LIN {X 0,Y 486.533,Z 891.187,A -85,B 0,C 180,E1 18755.175,E2 18755.175} C_VEL
LIN {X 0,Y 491.243,Z 865.57,A -85,B 0,C 180,E1 18754.171,E2 18754.171} C_VEL
LIN {X 0,Y 494.664,Z 842.648,A -85,B 0,C 180,E1 18753.45,E2 18753.45} C_VEL
LIN {X 0,Y 500.768,Z 797.276,A -85,B 0,C 180,E1 18752.327,E2 18752.327} C_VEL
LIN {X 0,Y 512.182,Z 708.591,A -85,B 0,C 180,E1 18750.377,E2 18750.377} C_VEL
LIN {X 0,Y 521.477,Z 628.395,A -85,B 0,C 180,E1 18748.797,E2 18748.797} C_VEL
LIN {X 0,Y 528.733,Z 554.168,A -85,B 0,C 180,E1 18747.473,E2 18747.473} C_VEL
LIN {X 0,Y 532.171,Z 510.95,A -85,B 0,C 180,E1 18746.749,E2 18746.749} C_VEL
LIN {X 0,Y 523.435,Z 503.495,A -85,B 0,C 180,E1 18744.489,E2 18744.489} C_VEL
LIN {X 0,Y 515.193,Z 497.011,A -85,B 0,C 180,E1 18742.118,E2 18742.118} C_VEL
LIN {X 0,Y 504.103,Z 489.409,A -85,B 0,C 180,E1 18738.384,E2 18738.384} C_VEL
LIN {X 0,Y 494.862,Z 485.329,A -85,B 0,C 180,E1 18734.51,E2 18734.51} C_VEL
LIN {X 0,Y 495.541,Z 486.097,A -85,B 0,C 180,E1 18730.345,E2 18730.345} C_VEL
LIN {X 0,Y 496.003,Z 486.953,A -85,B 0,C 180,E1 18728.93,E2 18728.93} C_VEL
LIN {X 0,Y 497.795,Z 491.194,A -85,B 0,C 180,E1 18724.955,E2 18724.955} C_VEL
LIN {X 0,Y 499.686,Z 495.798,A -85,B 0,C 180,E1 18722.064,E2 18722.064} C_VEL
LIN {X 0,Y 501.598,Z 500.282,A -85,B 0,C 180,E1 18719.772,E2 18719.772} C_VEL
LIN {X 0,Y 504.317,Z 506.652,A -85,B 0,C 180,E1 18717.045,E2 18717.045} C_VEL
LIN {X 0,Y 507.752,Z 515.364,A -85,B 0,C 180,E1 18714.009,E2 18714.009} C_VEL
LIN {X 0,Y 511.515,Z 525.152,A -85,B 0,C 180,E1 18711.116,E2 18711.116} C_VEL
LIN {X 0,Y 512.739,Z 529.148,A -85,B 0,C 180,E1 18710.119,E2 18710.119} C_VEL
LIN {X 0,Y 503.664,Z 561.52,A -85,B 0,C 180,E1 18707.086,E2 18707.086} C_VEL
LIN {X 0,Y 494.519,Z 596.305,A -85,B 0,C 180,E1 18703.918,E2 18703.918} C_VEL
LIN {X 0,Y 488.152,Z 622.653,A -85,B 0,C 180,E1 18701.597,E2 18701.597} C_VEL
LIN {X 0,Y 489.999,Z 648.401,A -85,B 0,C 180,E1 18699.881,E2 18699.881} C_VEL
LIN {X 0,Y 492.993,Z 672.9,A -85,B 0,C 180,E1 18698.025,E2 18698.025} C_VEL
LIN {X 0,Y 496.365,Z 691.421,A -85,B 0,C 180,E1 18696.441,E2 18696.441} C_VEL
LIN {X 0,Y 499.938,Z 706.73,A -85,B 0,C 180,E1 18695.023,E2 18695.023} C_VEL
LIN {X 0,Y 504.478,Z 722.336,A -85,B 0,C 180,E1 18693.452,E2 18693.452} C_VEL
LIN {X 0,Y 511.291,Z 740.682,A -85,B 0,C 180,E1 18691.419,E2 18691.419} C_VEL
LIN {X 0,Y 518.449,Z 755.933,A -85,B 0,C 180,E1 18689.569,E2 18689.569} C_VEL
LIN {X 0,Y 515.516,Z 776.629,A -85,B 0,C 180,E1 18689.383,E2 18689.383} C_VEL
LIN {X 0,Y 510.953,Z 813.16,A -85,B 0,C 180,E1 18688.666,E2 18688.666} C_VEL
LIN {X 0,Y 504.879,Z 851.472,A -85,B 0,C 180,E1 18687.765,E2 18687.765} C_VEL
LIN {X 0,Y 498.91,Z 884.135,A -85,B 0,C 180,E1 18686.793,E2 18686.793} C_VEL
LIN {X 0,Y 492.573,Z 916.172,A -85,B 0,C 180,E1 18685.602,E2 18685.602} C_VEL
LIN {X 0,Y 486.148,Z 946.544,A -85,B 0,C 180,E1 18684.229,E2 18684.229} C_VEL
LIN {X 0,Y 479.406,Z 976.457,A -85,B 0,C 180,E1 18682.618,E2 18682.618} C_VEL
LIN {X 0,Y 472.644,Z 1004.62,A -85,B 0,C 180,E1 18680.832,E2 18680.832} C_VEL
LIN {X 0,Y 466.937,Z 1026.075,A -85,B 0,C 180,E1 18679.222,E2 18679.222} C_VEL
LIN {X 0,Y 460.713,Z 1047.068,A -85,B 0,C 180,E1 18677.366,E2 18677.366} C_VEL
LIN {X 0,Y 454.254,Z 1066.808,A -85,B 0,C 180,E1 18675.311,E2 18675.311} C_VEL
LIN {X 0,Y 447.823,Z 1085.079,A -85,B 0,C 180,E1 18673.094,E2 18673.094} C_VEL
LIN {X 0,Y 441.211,Z 1102.891,A -85,B 0,C 180,E1 18670.57,E2 18670.57} C_VEL
LIN {X 0,Y 434.893,Z 1119.177,A -85,B 0,C 180,E1 18667.868,E2 18667.868} C_VEL
LIN {X 0,Y 428.995,Z 1134.014,A -85,B 0,C 180,E1 18664.983,E2 18664.983} C_VEL
LIN {X 0,Y 423.455,Z 1147.984,A -85,B 0,C 180,E1 18661.771,E2 18661.771} C_VEL
LIN {X 0,Y 418.686,Z 1160.386,A -85,B 0,C 180,E1 18658.373,E2 18658.373} C_VEL
LIN {X 0,Y 414.669,Z 1171.641,A -85,B 0,C 180,E1 18654.653,E2 18654.653} C_VEL
LIN {X 0,Y 411.75,Z 1180.908,A -85,B 0,C 180,E1 18650.912,E2 18650.912} C_VEL
LIN {X 0,Y 409.733,Z 1188.635,A -85,B 0,C 180,E1 18647.026,E2 18647.026} C_VEL
LIN {X 0,Y 408.63,Z 1194.443,A -85,B 0,C 180,E1 18643.296,E2 18643.296} C_VEL
LIN {X 0,Y 408.102,Z 1198.881,A -85,B 0,C 180,E1 18639.446,E2 18639.446} C_VEL
LIN {X 0,Y 407.951,Z 1201.616,A -85,B 0,C 180,E1 18635.907,E2 18635.907} C_VEL
LIN {X 0,Y 407.93,Z 1203.082,A -85,B 0,C 180,E1 18632.386,E2 18632.386} C_VEL
LIN {X 0,Y 407.934,Z 1203.299,A -85,B 0,C 180,E1 18628.875,E2 18628.875} C_VEL
LIN {X 0,Y 407.933,Z 1202.268,A -85,B 0,C 180,E1 18625.359,E2 18625.359} C_VEL
LIN {X 0,Y 408.025,Z 1199.983,A -85,B 0,C 180,E1 18621.827,E2 18621.827} C_VEL
LIN {X 0,Y 408.369,Z 1196.238,A -85,B 0,C 180,E1 18618.129,E2 18618.129} C_VEL
LIN {X 0,Y 409.239,Z 1191.031,A -85,B 0,C 180,E1 18614.408,E2 18614.408} C_VEL
LIN {X 0,Y 410.895,Z 1183.951,A -85,B 0,C 180,E1 18610.524,E2 18610.524} C_VEL
LIN {X 0,Y 413.414,Z 1175.392,A -85,B 0,C 180,E1 18606.78,E2 18606.78} C_VEL
LIN {X 0,Y 416.887,Z 1165.252,A -85,B 0,C 180,E1 18603.155,E2 18603.155} C_VEL
LIN {X 0,Y 421.135,Z 1153.9,A -85,B 0,C 180,E1 18599.777,E2 18599.777} C_VEL
LIN {X 0,Y 426.483,Z 1140.338,A -85,B 0,C 180,E1 18596.405,E2 18596.405} C_VEL
LIN {X 0,Y 432.262,Z 1125.794,A -85,B 0,C 180,E1 18593.358,E2 18593.358} C_VEL
LIN {X 0,Y 438.608,Z 1109.68,A -85,B 0,C 180,E1 18590.502,E2 18590.502} C_VEL
LIN {X 0,Y 444.992,Z 1092.865,A -85,B 0,C 180,E1 18587.962,E2 18587.962} C_VEL
LIN {X 0,Y 451.682,Z 1074.286,A -85,B 0,C 180,E1 18585.561,E2 18585.561} C_VEL
LIN {X 0,Y 458.264,Z 1054.685,A -85,B 0,C 180,E1 18583.399,E2 18583.399} C_VEL
LIN {X 0,Y 464.518,Z 1034.442,A -85,B 0,C 180,E1 18581.488,E2 18581.488} C_VEL
LIN {X 0,Y 470.519,Z 1012.971,A -85,B 0,C 180,E1 18579.766,E2 18579.766} C_VEL
LIN {X 0,Y 476.328,Z 989.375,A -85,B 0,C 180,E1 18578.173,E2 18578.173} C_VEL
LIN {X 0,Y 482.582,Z 962.508,A -85,B 0,C 180,E1 18576.602,E2 18576.602} C_VEL
LIN {X 0,Y 489.045,Z 932.988,A -85,B 0,C 180,E1 18575.131,E2 18575.131} C_VEL
LIN {X 0,Y 495.498,Z 901.478,A -85,B 0,C 180,E1 18573.824,E2 18573.824} C_VEL
LIN {X 0,Y 501.919,Z 867.701,A -85,B 0,C 180,E1 18572.694,E2 18572.694} C_VEL
LIN {X 0,Y 508.145,Z 831.765,A -85,B 0,C 180,E1 18571.754,E2 18571.754} C_VEL
LIN {X 0,Y 513.646,Z 791.804,A -85,B 0,C 180,E1 18570.894,E2 18570.894} C_VEL
LIN {X 0,Y 517.57,Z 753.556,A -85,B 0,C 180,E1 18570.212,E2 18570.212} C_VEL
LIN {X 0,Y 522.49,Z 683.228,A -85,B 0,C 180,E1 18569.21,E2 18569.21} C_VEL
LIN {X 0,Y 524.513,Z 660.576,A -85,B 0,C 180,E1 18568.918,E2 18568.918} C_VEL
LIN {X 0,Y 529.301,Z 622.998,A -85,B 0,C 180,E1 18568.284,E2 18568.284} C_VEL
LIN {X 0,Y 531.877,Z 604.095,A -85,B 0,C 180,E1 18567.995,E2 18567.995} C_VEL
LIN {X 0,Y 536.492,Z 568.871,A -85,B 0,C 180,E1 18567.424,E2 18567.424} C_VEL
LIN {X 0,Y 539.728,Z 546.528,A -85,B 0,C 180,E1 18567.12,E2 18567.12} C_VEL
LIN {X 0,Y 543.093,Z 519.32,A -85,B 0,C 180,E1 18566.641,E2 18566.641} C_VEL
LIN {X 0,Y 533.557,Z 502.875,A -85,B 0,C 180,E1 18563.966,E2 18563.966} C_VEL
LIN {X 0,Y 527.481,Z 493.209,A -85,B 0,C 180,E1 18562.103,E2 18562.103} C_VEL
LIN {X 0,Y 525.221,Z 498.395,A -85,B 0,C 180,E1 18561.814,E2 18561.814} C_VEL
LIN {X 0,Y 519.364,Z 513.075,A -85,B 0,C 180,E1 18561.101,E2 18561.101} C_VEL
LIN {X 0,Y 515.098,Z 522.888,A -85,B 0,C 180,E1 18560.511,E2 18560.511} C_VEL
LIN {X 0,Y 509.416,Z 537.56,A -85,B 0,C 180,E1 18559.776,E2 18559.776} C_VEL
LIN {X 0,Y 505.389,Z 547.114,A -85,B 0,C 180,E1 18559.181,E2 18559.181} C_VEL
LIN {X 0,Y 499.874,Z 561.958,A -85,B 0,C 180,E1 18558.432,E2 18558.432} C_VEL
LIN {X 0,Y 495.743,Z 572.106,A -85,B 0,C 180,E1 18557.78,E2 18557.78} C_VEL
LIN {X 0,Y 490.352,Z 587.299,A -85,B 0,C 180,E1 18557.011,E2 18557.011} C_VEL
LIN {X 0,Y 485.983,Z 598.469,A -85,B 0,C 180,E1 18556.272,E2 18556.272} C_VEL
LIN {X 0,Y 482.289,Z 610.977,A -85,B 0,C 180,E1 18555.674,E2 18555.674} C_VEL
LIN {X 0,Y 478.187,Z 626.414,A -85,B 0,C 180,E1 18554.749,E2 18554.749} C_VEL
LIN {X 0,Y 476.998,Z 630.964,A -85,B 0,C 180,E1 18554.471,E2 18554.471} C_VEL
LIN {X 0,Y 472.235,Z 652.376,A -85,B 0,C 180,E1 18553.476,E2 18553.476} C_VEL
LIN {X 0,Y 468.085,Z 669.271,A -85,B 0,C 180,E1 18552.467,E2 18552.467} C_VEL
LIN {X 0,Y 466.576,Z 674.939,A -85,B 0,C 180,E1 18552.1,E2 18552.1} C_VEL
LIN {X 0,Y 461.683,Z 695.246,A -85,B 0,C 180,E1 18551.113,E2 18551.113} C_VEL
LIN {X 0,Y 457.616,Z 709.605,A -85,B 0,C 180,E1 18550.178,E2 18550.178} C_VEL
LIN {X 0,Y 456.259,Z 714.146,A -85,B 0,C 180,E1 18549.858,E2 18549.858} C_VEL
LIN {X 0,Y 451.518,Z 731.526,A -85,B 0,C 180,E1 18548.959,E2 18548.959} C_VEL
LIN {X 0,Y 447.932,Z 743.114,A -85,B 0,C 180,E1 18548.133,E2 18548.133} C_VEL
LIN {X 0,Y 446.662,Z 747.062,A -85,B 0,C 180,E1 18547.824,E2 18547.824} C_VEL
LIN {X 0,Y 441.934,Z 763.035,A -85,B 0,C 180,E1 18546.936,E2 18546.936} C_VEL
LIN {X 0,Y 438.611,Z 773.144,A -85,B 0,C 180,E1 18546.133,E2 18546.133} C_VEL
LIN {X 0,Y 437.676,Z 775.933,A -85,B 0,C 180,E1 18545.909,E2 18545.909} C_VEL
LIN {X 0,Y 433.17,Z 790.556,A -85,B 0,C 180,E1 18545.049,E2 18545.049} C_VEL
LIN {X 0,Y 430.208,Z 799.346,A -85,B 0,C 180,E1 18544.295,E2 18544.295} C_VEL
LIN {X 0,Y 429.367,Z 801.766,A -85,B 0,C 180,E1 18544.076,E2 18544.076} C_VEL
LIN {X 0,Y 425.227,Z 814.86,A -85,B 0,C 180,E1 18543.286,E2 18543.286} C_VEL
LIN {X 0,Y 422.513,Z 823.016,A -85,B 0,C 180,E1 18542.56,E2 18542.56} C_VEL
LIN {X 0,Y 421.861,Z 825.173,A -85,B 0,C 180,E1 18542.309,E2 18542.309} C_VEL
LIN {X 0,Y 420.52,Z 859.932,A -85,B 0,C 180,E1 18540.647,E2 18540.647} C_VEL
LIN {X 0,Y 418.335,Z 883.831,A -85,B 0,C 180,E1 18539.619,E2 18539.619} C_VEL
LIN {X 0,Y 416.068,Z 978.523,A -85,B 0,C 180,E1 18537.607,E2 18537.607} C_VEL
LIN {X 0,Y 416.149,Z 999.978,A -85,B 0,C 180,E1 18537.078,E2 18537.078} C_VEL
LIN {X 0,Y 416.065,Z 1014.863,A -85,B 0,C 180,E1 18536.487,E2 18536.487} C_VEL
LIN {X 0,Y 415.715,Z 1027.895,A -85,B 0,C 180,E1 18535.724,E2 18535.724} C_VEL
LIN {X 0,Y 415.303,Z 1039.006,A -85,B 0,C 180,E1 18534.889,E2 18534.889} C_VEL
LIN {X 0,Y 414.72,Z 1050.801,A -85,B 0,C 180,E1 18533.771,E2 18533.771} C_VEL
LIN {X 0,Y 413.977,Z 1061.496,A -85,B 0,C 180,E1 18532.446,E2 18532.446} C_VEL
LIN {X 0,Y 413.353,Z 1069.351,A -85,B 0,C 180,E1 18531.234,E2 18531.234} C_VEL
LIN {X 0,Y 412.756,Z 1076.09,A -85,B 0,C 180,E1 18529.955,E2 18529.955} C_VEL
LIN {X 0,Y 412.168,Z 1082.093,A -85,B 0,C 180,E1 18528.526,E2 18528.526} C_VEL
LIN {X 0,Y 411.599,Z 1087.594,A -85,B 0,C 180,E1 18526.8,E2 18526.8} C_VEL
LIN {X 0,Y 411.113,Z 1091.473,A -85,B 0,C 180,E1 18524.916,E2 18524.916} C_VEL
LIN {X 0,Y 410.832,Z 1093.388,A -85,B 0,C 180,E1 18523.31,E2 18523.31} C_VEL
LIN {X 0,Y 410.662,Z 1094.056,A -85,B 0,C 180,E1 18521.694,E2 18521.694} C_VEL
LIN {X 0,Y 410.596,Z 1093.471,A -85,B 0,C 180,E1 18520.053,E2 18520.053} C_VEL
LIN {X 0,Y 410.66,Z 1091.119,A -85,B 0,C 180,E1 18518.077,E2 18518.077} C_VEL
LIN {X 0,Y 410.869,Z 1086.998,A -85,B 0,C 180,E1 18516.212,E2 18516.212} C_VEL
LIN {X 0,Y 411.162,Z 1082.209,A -85,B 0,C 180,E1 18514.659,E2 18514.659} C_VEL
LIN {X 0,Y 411.625,Z 1075.463,A -85,B 0,C 180,E1 18512.983,E2 18512.983} C_VEL
LIN {X 0,Y 412.258,Z 1066.079,A -85,B 0,C 180,E1 18511.219,E2 18511.219} C_VEL
LIN {X 0,Y 412.825,Z 1057.298,A -85,B 0,C 180,E1 18509.909,E2 18509.909} C_VEL
LIN {X 0,Y 413.474,Z 1046.64,A -85,B 0,C 180,E1 18508.613,E2 18508.613} C_VEL
LIN {X 0,Y 414.125,Z 1033.201,A -85,B 0,C 180,E1 18507.341,E2 18507.341} C_VEL
LIN {X 0,Y 414.589,Z 1021.462,A -85,B 0,C 180,E1 18506.475,E2 18506.475} C_VEL
LIN {X 0,Y 414.947,Z 1008.747,A -85,B 0,C 180,E1 18505.745,E2 18505.745} C_VEL
LIN {X 0,Y 415.145,Z 998.499,A -85,B 0,C 180,E1 18505.276,E2 18505.276} C_VEL
LIN {X 0,Y 416.23,Z 998.976,A -85,B 0,C 180,E1 18504.96,E2 18504.96} C_VEL
LIN {X 0,Y 418.224,Z 998.373,A -85,B 0,C 180,E1 18504.649,E2 18504.649} C_VEL
LIN {X 0,Y 421.758,Z 996.071,A -85,B 0,C 180,E1 18504.323,E2 18504.323} C_VEL
LIN {X 0,Y 425.485,Z 994.503,A -85,B 0,C 180,E1 18503.853,E2 18503.853} C_VEL
LIN {X 0,Y 429.216,Z 991.915,A -85,B 0,C 180,E1 18503.555,E2 18503.555} C_VEL
LIN {X 0,Y 433.245,Z 989.836,A -85,B 0,C 180,E1 18503.126,E2 18503.126} C_VEL
LIN {X 0,Y 437.995,Z 986.45,A -85,B 0,C 180,E1 18502.774,E2 18502.774} C_VEL
LIN {X 0,Y 443.74,Z 982.814,A -85,B 0,C 180,E1 18502.273,E2 18502.273} C_VEL
LIN {X 0,Y 448.015,Z 979.633,A -85,B 0,C 180,E1 18501.976,E2 18501.976} C_VEL
LIN {X 0,Y 453.582,Z 975.703,A -85,B 0,C 180,E1 18501.563,E2 18501.563} C_VEL
LIN {X 0,Y 457.655,Z 972.4,A -85,B 0,C 180,E1 18501.328,E2 18501.328} C_VEL
LIN {X 0,Y 464.355,Z 967.489,A -85,B 0,C 180,E1 18500.882,E2 18500.882} C_VEL
LIN {X 0,Y 469.177,Z 963.473,A -85,B 0,C 180,E1 18500.613,E2 18500.613} C_VEL
LIN {X 0,Y 462.39,Z 987.036,A -85,B 0,C 180,E1 18498.735,E2 18498.735} C_VEL
LIN {X 0,Y 455.753,Z 1008.668,A -85,B 0,C 180,E1 18496.752,E2 18496.752} C_VEL
LIN {X 0,Y 448.811,Z 1029.862,A -85,B 0,C 180,E1 18494.481,E2 18494.481} C_VEL
LIN {X 0,Y 442.19,Z 1049.901,A -85,B 0,C 180,E1 18492.016,E2 18492.016} C_VEL
LIN {X 0,Y 435.89,Z 1068.357,A -85,B 0,C 180,E1 18489.371,E2 18489.371} C_VEL
LIN {X 0,Y 430.062,Z 1085.804,A -85,B 0,C 180,E1 18486.528,E2 18486.528} C_VEL
LIN {X 0,Y 424.875,Z 1101.35,A -85,B 0,C 180,E1 18483.577,E2 18483.577} C_VEL
LIN {X 0,Y 420.599,Z 1115.061,A -85,B 0,C 180,E1 18480.617,E2 18480.617} C_VEL
LIN {X 0,Y 416.519,Z 1128.903,A -85,B 0,C 180,E1 18477.138,E2 18477.138} C_VEL
LIN {X 0,Y 413.879,Z 1138.826,A -85,B 0,C 180,E1 18474.25,E2 18474.25} C_VEL
LIN {X 0,Y 411.493,Z 1149.153,A -85,B 0,C 180,E1 18470.781,E2 18470.781} C_VEL
LIN {X 0,Y 409.837,Z 1157.541,A -85,B 0,C 180,E1 18467.318,E2 18467.318} C_VEL
LIN {X 0,Y 408.929,Z 1163.444,A -85,B 0,C 180,E1 18464.387,E2 18464.387} C_VEL
LIN {X 0,Y 407.715,Z 1165.443,A -85,B 0,C 180,E1 18463.346,E2 18463.346} C_VEL
LIN {X 0,Y 400.802,Z 1170.209,A -85,B 0,C 180,E1 18460.402,E2 18460.402} C_VEL
LIN {X 0,Y 400.183,Z 1171.12,A -85,B 0,C 180,E1 18459.621,E2 18459.621} C_VEL
LIN {X 0,Y 400.01,Z 1173.979,A -85,B 0,C 180,E1 18456.749,E2 18456.749} C_VEL
LIN {X 0,Y 399.949,Z 1175.778,A -85,B 0,C 180,E1 18454.016,E2 18454.016} C_VEL
LIN {X 0,Y 399.937,Z 1176.672,A -85,B 0,C 180,E1 18451.291,E2 18451.291} C_VEL
LIN {X 0,Y 399.936,Z 1176.664,A -85,B 0,C 180,E1 18448.569,E2 18448.569} C_VEL
LIN {X 0,Y 399.951,Z 1175.753,A -85,B 0,C 180,E1 18445.844,E2 18445.844} C_VEL
LIN {X 0,Y 400.011,Z 1173.938,A -85,B 0,C 180,E1 18443.111,E2 18443.111} C_VEL
LIN {X 0,Y 400.189,Z 1171.042,A -85,B 0,C 180,E1 18440.22,E2 18440.22} C_VEL
LIN {X 0,Y 400.686,Z 1166.243,A -85,B 0,C 180,E1 18436.713,E2 18436.713} C_VEL
LIN {X 0,Y 401.628,Z 1159.776,A -85,B 0,C 180,E1 18433.216,E2 18433.216} C_VEL
LIN {X 0,Y 402.974,Z 1152.797,A -85,B 0,C 180,E1 18430.12,E2 18430.12} C_VEL
LIN {X 0,Y 404.869,Z 1144.61,A -85,B 0,C 180,E1 18427.035,E2 18427.035} C_VEL
LIN {X 0,Y 408.119,Z 1132.508,A -85,B 0,C 180,E1 18423.207,E2 18423.207} C_VEL
LIN {X 0,Y 411.478,Z 1121.236,A -85,B 0,C 180,E1 18420.171,E2 18420.171} C_VEL
LIN {X 0,Y 416.221,Z 1106.792,A -85,B 0,C 180,E1 18416.792,E2 18416.792} C_VEL
LIN {X 0,Y 421.223,Z 1091.936,A -85,B 0,C 180,E1 18413.812,E2 18413.812} C_VEL
LIN {X 0,Y 426.979,Z 1075.735,A -85,B 0,C 180,E1 18410.957,E2 18410.957} C_VEL
LIN {X 0,Y 433.411,Z 1057.452,A -85,B 0,C 180,E1 18408.188,E2 18408.188} C_VEL
LIN {X 0,Y 439.516,Z 1040.153,A -85,B 0,C 180,E1 18405.885,E2 18405.885} C_VEL
LIN {X 0,Y 446.769,Z 1018.866,A -85,B 0,C 180,E1 18403.431,E2 18403.431} C_VEL
LIN {X 0,Y 453.158,Z 999.494,A -85,B 0,C 180,E1 18401.49,E2 18401.49} C_VEL
LIN {X 0,Y 460.44,Z 976.023,A -85,B 0,C 180,E1 18399.47,E2 18399.47} C_VEL
LIN {X 0,Y 466.465,Z 955.22,A -85,B 0,C 180,E1 18397.928,E2 18397.928} C_VEL
LIN {X 0,Y 473.017,Z 930.366,A -85,B 0,C 180,E1 18396.357,E2 18396.357} C_VEL
LIN {X 0,Y 477.985,Z 909.341,A -85,B 0,C 180,E1 18395.23,E2 18395.23} C_VEL
LIN {X 0,Y 483.181,Z 884.732,A -85,B 0,C 180,E1 18394.112,E2 18394.112} C_VEL
LIN {X 0,Y 487.366,Z 861.137,A -85,B 0,C 180,E1 18393.24,E2 18393.24} C_VEL
LIN {X 0,Y 491.222,Z 835.424,A -85,B 0,C 180,E1 18392.469,E2 18392.469} C_VEL
LIN {X 0,Y 503.581,Z 744.719,A -85,B 0,C 180,E1 18390.359,E2 18390.359} C_VEL
LIN {X 0,Y 513.783,Z 663.571,A -85,B 0,C 180,E1 18388.681,E2 18388.681} C_VEL
LIN {X 0,Y 522.016,Z 587.861,A -85,B 0,C 180,E1 18387.273,E2 18387.273} C_VEL
LIN {X 0,Y 528.229,Z 517.228,A -85,B 0,C 180,E1 18386.077,E2 18386.077} C_VEL
LIN {X 0,Y 528.189,Z 516.76,A -85,B 0,C 180,E1 18386.052,E2 18386.052} C_VEL
LIN {X 0,Y 521.537,Z 511.047,A -85,B 0,C 180,E1 18384.283,E2 18384.283} C_VEL
LIN {X 0,Y 513.386,Z 504.608,A -85,B 0,C 180,E1 18381.899,E2 18381.899} C_VEL
LIN {X 0,Y 502.868,Z 497.289,A -85,B 0,C 180,E1 18378.31,E2 18378.31} C_VEL
LIN {X 0,Y 493.62,Z 493.235,A -85,B 0,C 180,E1 18374.427,E2 18374.427} C_VEL
LIN {X 0,Y 490.745,Z 492.243,A -85,B 0,C 180,E1 18372.951,E2 18372.951} C_VEL
LIN {X 0,Y 491.759,Z 493.451,A -85,B 0,C 180,E1 18369.244,E2 18369.244} C_VEL
LIN {X 0,Y 493.518,Z 497.984,A -85,B 0,C 180,E1 18364.998,E2 18364.998} C_VEL
LIN {X 0,Y 495.306,Z 502.39,A -85,B 0,C 180,E1 18362.198,E2 18362.198} C_VEL
LIN {X 0,Y 497.174,Z 506.879,A -85,B 0,C 180,E1 18359.885,E2 18359.885} C_VEL
LIN {X 0,Y 499.729,Z 512.968,A -85,B 0,C 180,E1 18357.248,E2 18357.248} C_VEL
LIN {X 0,Y 503.08,Z 521.676,A -85,B 0,C 180,E1 18354.182,E2 18354.182} C_VEL
LIN {X 0,Y 506.762,Z 531.481,A -85,B 0,C 180,E1 18351.261,E2 18351.261} C_VEL
LIN {X 0,Y 507.584,Z 534.086,A -85,B 0,C 180,E1 18350.59,E2 18350.59} C_VEL
LIN {X 0,Y 498.418,Z 565.826,A -85,B 0,C 180,E1 18347.605,E2 18347.605} C_VEL
LIN {X 0,Y 488.94,Z 600.817,A -85,B 0,C 180,E1 18344.4,E2 18344.4} C_VEL
LIN {X 0,Y 485.065,Z 616.581,A -85,B 0,C 180,E1 18343.007,E2 18343.007} C_VEL
LIN {X 0,Y 486.674,Z 645.609,A -85,B 0,C 180,E1 18341.089,E2 18341.089} C_VEL
LIN {X 0,Y 488.765,Z 667.497,A -85,B 0,C 180,E1 18339.492,E2 18339.492} C_VEL
LIN {X 0,Y 492.052,Z 689.916,A -85,B 0,C 180,E1 18337.666,E2 18337.666} C_VEL
LIN {X 0,Y 496.427,Z 710.604,A -85,B 0,C 180,E1 18335.755,E2 18335.755} C_VEL
LIN {X 0,Y 501.181,Z 727.72,A -85,B 0,C 180,E1 18334.013,E2 18334.013} C_VEL
LIN {X 0,Y 507.875,Z 746.427,A -85,B 0,C 180,E1 18331.915,E2 18331.915} C_VEL
LIN {X 0,Y 513.758,Z 759.555,A -85,B 0,C 180,E1 18330.311,E2 18330.311} C_VEL
LIN {X 0,Y 510.892,Z 779.529,A -85,B 0,C 180,E1 18330.097,E2 18330.097} C_VEL
LIN {X 0,Y 505.749,Z 818.706,A -85,B 0,C 180,E1 18329.3,E2 18329.3} C_VEL
LIN {X 0,Y 499.219,Z 857.054,A -85,B 0,C 180,E1 18328.363,E2 18328.363} C_VEL
LIN {X 0,Y 492.909,Z 890.183,A -85,B 0,C 180,E1 18327.332,E2 18327.332} C_VEL
LIN {X 0,Y 486.371,Z 922.041,A -85,B 0,C 180,E1 18326.099,E2 18326.099} C_VEL
LIN {X 0,Y 479.461,Z 953.461,A -85,B 0,C 180,E1 18324.624,E2 18324.624} C_VEL
LIN {X 0,Y 472.37,Z 983.55,A -85,B 0,C 180,E1 18322.937,E2 18322.937} C_VEL
LIN {X 0,Y 465.742,Z 1009.903,A -85,B 0,C 180,E1 18321.194,E2 18321.194} C_VEL
LIN {X 0,Y 459.37,Z 1032.171,A -85,B 0,C 180,E1 18319.43,E2 18319.43} C_VEL
LIN {X 0,Y 452.871,Z 1052.669,A -85,B 0,C 180,E1 18317.51,E2 18317.51} C_VEL
LIN {X 0,Y 446.067,Z 1072.391,A -85,B 0,C 180,E1 18315.346,E2 18315.346} C_VEL
LIN {X 0,Y 439.188,Z 1090.996,A -85,B 0,C 180,E1 18312.953,E2 18312.953} C_VEL
LIN {X 0,Y 432.761,Z 1107.475,A -85,B 0,C 180,E1 18310.482,E2 18310.482} C_VEL
LIN {X 0,Y 426.092,Z 1123.874,A -85,B 0,C 180,E1 18307.596,E2 18307.596} C_VEL
LIN {X 0,Y 419.948,Z 1138.652,A -85,B 0,C 180,E1 18304.516,E2 18304.516} C_VEL
LIN {X 0,Y 414.52,Z 1151.912,A -85,B 0,C 180,E1 18301.237,E2 18301.237} C_VEL
LIN {X 0,Y 409.881,Z 1163.689,A -85,B 0,C 180,E1 18297.769,E2 18297.769} C_VEL
LIN {X 0,Y 406.15,Z 1173.986,A -85,B 0,C 180,E1 18294.119,E2 18294.119} C_VEL
LIN {X 0,Y 403.355,Z 1182.79,A -85,B 0,C 180,E1 18290.305,E2 18290.305} C_VEL
LIN {X 0,Y 401.53,Z 1189.848,A -85,B 0,C 180,E1 18286.49,E2 18286.49} C_VEL
LIN {X 0,Y 400.504,Z 1195.302,A -85,B 0,C 180,E1 18282.689,E2 18282.689} C_VEL
LIN {X 0,Y 400.067,Z 1199.269,A -85,B 0,C 180,E1 18278.912,E2 18278.912} C_VEL
LIN {X 0,Y 399.944,Z 1201.754,A -85,B 0,C 180,E1 18275.306,E2 18275.306} C_VEL
LIN {X 0,Y 399.934,Z 1202.969,A -85,B 0,C 180,E1 18271.861,E2 18271.861} C_VEL
LIN {X 0,Y 399.936,Z 1202.996,A -85,B 0,C 180,E1 18268.422,E2 18268.422} C_VEL
LIN {X 0,Y 399.942,Z 1201.821,A -85,B 0,C 180,E1 18264.835,E2 18264.835} C_VEL
LIN {X 0,Y 400.057,Z 1199.39,A -85,B 0,C 180,E1 18261.229,E2 18261.229} C_VEL
LIN {X 0,Y 400.48,Z 1195.481,A -85,B 0,C 180,E1 18257.453,E2 18257.453} C_VEL
LIN {X 0,Y 401.483,Z 1190.086,A -85,B 0,C 180,E1 18253.653,E2 18253.653} C_VEL
LIN {X 0,Y 403.357,Z 1182.785,A -85,B 0,C 180,E1 18249.692,E2 18249.692} C_VEL
LIN {X 0,Y 406.155,Z 1173.978,A -85,B 0,C 180,E1 18245.877,E2 18245.877} C_VEL
LIN {X 0,Y 409.884,Z 1163.678,A -85,B 0,C 180,E1 18242.228,E2 18242.228} C_VEL
LIN {X 0,Y 414.525,Z 1151.898,A -85,B 0,C 180,E1 18238.76,E2 18238.76} C_VEL
LIN {X 0,Y 419.983,Z 1138.549,A -85,B 0,C 180,E1 18235.463,E2 18235.463} C_VEL
LIN {X 0,Y 426.095,Z 1123.839,A -85,B 0,C 180,E1 18232.4,E2 18232.4} C_VEL
LIN {X 0,Y 432.919,Z 1107.068,A -85,B 0,C 180,E1 18229.453,E2 18229.453} C_VEL
LIN {X 0,Y 439.809,Z 1089.346,A -85,B 0,C 180,E1 18226.817,E2 18226.817} C_VEL
LIN {X 0,Y 446.713,Z 1070.541,A -85,B 0,C 180,E1 18224.435,E2 18224.435} C_VEL
LIN {X 0,Y 453.503,Z 1050.665,A -85,B 0,C 180,E1 18222.291,E2 18222.291} C_VEL
LIN {X 0,Y 460.049,Z 1029.72,A -85,B 0,C 180,E1 18220.368,E2 18220.368} C_VEL
LIN {X 0,Y 466.198,Z 1007.987,A -85,B 0,C 180,E1 18218.674,E2 18218.674} C_VEL
LIN {X 0,Y 472.604,Z 982.271,A -85,B 0,C 180,E1 18216.995,E2 18216.995} C_VEL
LIN {X 0,Y 480.508,Z 948.58,A -85,B 0,C 180,E1 18215.134,E2 18215.134} C_VEL
LIN {X 0,Y 487.354,Z 917.154,A -85,B 0,C 180,E1 18213.699,E2 18213.699} C_VEL
LIN {X 0,Y 493.983,Z 884.599,A -85,B 0,C 180,E1 18212.481,E2 18212.481} C_VEL
LIN {X 0,Y 500.295,Z 850.881,A -85,B 0,C 180,E1 18211.477,E2 18211.477} C_VEL
LIN {X 0,Y 506.6,Z 812.409,A -85,B 0,C 180,E1 18210.565,E2 18210.565} C_VEL
LIN {X 0,Y 511.799,Z 770.225,A -85,B 0,C 180,E1 18209.724,E2 18209.724} C_VEL
LIN {X 0,Y 515.455,Z 728.545,A -85,B 0,C 180,E1 18209.06,E2 18209.06} C_VEL
LIN {X 0,Y 519.991,Z 665.837,A -85,B 0,C 180,E1 18208.233,E2 18208.233} C_VEL
LIN {X 0,Y 523.25,Z 637.808,A -85,B 0,C 180,E1 18207.755,E2 18207.755} C_VEL
LIN {X 0,Y 527.822,Z 604.692,A -85,B 0,C 180,E1 18207.252,E2 18207.252} C_VEL
LIN {X 0,Y 532.553,Z 569.137,A -85,B 0,C 180,E1 18206.678,E2 18206.678} C_VEL
LIN {X 0,Y 535.805,Z 546.906,A -85,B 0,C 180,E1 18206.377,E2 18206.377} C_VEL
LIN {X 0,Y 538.738,Z 523.81,A -85,B 0,C 180,E1 18205.977,E2 18205.977} C_VEL
LIN {X 0,Y 529.802,Z 508.232,A -85,B 0,C 180,E1 18203.379,E2 18203.379} C_VEL
LIN {X 0,Y 526.894,Z 503.656,A -85,B 0,C 180,E1 18202.482,E2 18202.482} C_VEL
LIN {X 0,Y 520.808,Z 518.492,A -85,B 0,C 180,E1 18201.749,E2 18201.749} C_VEL
LIN {X 0,Y 517.074,Z 526.968,A -85,B 0,C 180,E1 18201.247,E2 18201.247} C_VEL
LIN {X 0,Y 511.134,Z 542.014,A -85,B 0,C 180,E1 18200.497,E2 18200.497} C_VEL
LIN {X 0,Y 507.188,Z 551.271,A -85,B 0,C 180,E1 18199.934,E2 18199.934} C_VEL
LIN {X 0,Y 501.482,Z 566.318,A -85,B 0,C 180,E1 18199.177,E2 18199.177} C_VEL
LIN {X 0,Y 497.408,Z 576.197,A -85,B 0,C 180,E1 18198.557,E2 18198.557} C_VEL
LIN {X 0,Y 491.817,Z 591.617,A -85,B 0,C 180,E1 18197.779,E2 18197.779} C_VEL
LIN {X 0,Y 487.471,Z 602.573,A -85,B 0,C 180,E1 18197.071,E2 18197.071} C_VEL
LIN {X 0,Y 483.811,Z 614.811,A -85,B 0,C 180,E1 18196.489,E2 18196.489} C_VEL
LIN {X 0,Y 479.476,Z 630.68,A -85,B 0,C 180,E1 18195.544,E2 18195.544} C_VEL
LIN {X 0,Y 478.37,Z 634.918,A -85,B 0,C 180,E1 18195.301,E2 18195.301} C_VEL
LIN {X 0,Y 473.456,Z 656.393,A -85,B 0,C 180,E1 18194.306,E2 18194.306} C_VEL
LIN {X 0,Y 469.127,Z 673.437,A -85,B 0,C 180,E1 18193.293,E2 18193.293} C_VEL
LIN {X 0,Y 467.664,Z 678.834,A -85,B 0,C 180,E1 18192.958,E2 18192.958} C_VEL
LIN {X 0,Y 462.588,Z 699.243,A -85,B 0,C 180,E1 18191.968,E2 18191.968} C_VEL
LIN {X 0,Y 458.259,Z 713.975,A -85,B 0,C 180,E1 18191.013,E2 18191.013} C_VEL
LIN {X 0,Y 456.968,Z 718.237,A -85,B 0,C 180,E1 18190.732,E2 18190.732} C_VEL
LIN {X 0,Y 451.998,Z 735.866,A -85,B 0,C 180,E1 18189.815,E2 18189.815} C_VEL
LIN {X 0,Y 448.177,Z 747.722,A -85,B 0,C 180,E1 18188.969,E2 18188.969} C_VEL
LIN {X 0,Y 447.018,Z 751.288,A -85,B 0,C 180,E1 18188.712,E2 18188.712} C_VEL
LIN {X 0,Y 442.098,Z 767.347,A -85,B 0,C 180,E1 18187.814,E2 18187.814} C_VEL
LIN {X 0,Y 438.48,Z 777.882,A -85,B 0,C 180,E1 18186.975,E2 18186.975} C_VEL
LIN {X 0,Y 436.744,Z 783.34,A -85,B 0,C 180,E1 18186.653,E2 18186.653} C_VEL
LIN {X 0,Y 432.228,Z 797.15,A -85,B 0,C 180,E1 18185.775,E2 18185.775} C_VEL
LIN {X 0,Y 429.109,Z 805.975,A -85,B 0,C 180,E1 18185.005,E2 18185.005} C_VEL
LIN {X 0,Y 424.802,Z 819.185,A -85,B 0,C 180,E1 18184.195,E2 18184.195} C_VEL
LIN {X 0,Y 421.775,Z 827.775,A -85,B 0,C 180,E1 18183.428,E2 18183.428} C_VEL
LIN {X 0,Y 420.968,Z 830.07,A -85,B 0,C 180,E1 18183.221,E2 18183.221} C_VEL
LIN {X 0,Y 416.812,Z 842.6,A -85,B 0,C 180,E1 18182.423,E2 18182.423} C_VEL
LIN {X 0,Y 414.266,Z 849.824,A -85,B 0,C 180,E1 18181.729,E2 18181.729} C_VEL
LIN {X 0,Y 413.752,Z 851.556,A -85,B 0,C 180,E1 18181.523,E2 18181.523} C_VEL
LIN {X 0,Y 412.473,Z 868.78,A -85,B 0,C 180,E1 18180.729,E2 18180.729} C_VEL
LIN {X 0,Y 410.937,Z 885.131,A -85,B 0,C 180,E1 18180.027,E2 18180.027} C_VEL
LIN {X 0,Y 408.524,Z 978.565,A -85,B 0,C 180,E1 18177.979,E2 18177.979} C_VEL
LIN {X 0,Y 408.593,Z 1001.02,A -85,B 0,C 180,E1 18177.418,E2 18177.418} C_VEL
LIN {X 0,Y 408.508,Z 1015.45,A -85,B 0,C 180,E1 18176.843,E2 18176.843} C_VEL
LIN {X 0,Y 408.141,Z 1028.655,A -85,B 0,C 180,E1 18176.067,E2 18176.067} C_VEL
LIN {X 0,Y 407.692,Z 1039.793,A -85,B 0,C 180,E1 18175.217,E2 18175.217} C_VEL
LIN {X 0,Y 407.093,Z 1051.067,A -85,B 0,C 180,E1 18174.134,E2 18174.134} C_VEL
LIN {X 0,Y 406.262,Z 1062.664,A -85,B 0,C 180,E1 18172.692,E2 18172.692} C_VEL
LIN {X 0,Y 405.623,Z 1070.328,A -85,B 0,C 180,E1 18171.494,E2 18171.494} C_VEL
LIN {X 0,Y 404.991,Z 1077.115,A -85,B 0,C 180,E1 18170.191,E2 18170.191} C_VEL
LIN {X 0,Y 404.424,Z 1082.607,A -85,B 0,C 180,E1 18168.881,E2 18168.881} C_VEL
LIN {X 0,Y 403.889,Z 1087.41,A -85,B 0,C 180,E1 18167.417,E2 18167.417} C_VEL
LIN {X 0,Y 403.392,Z 1091.629,A -85,B 0,C 180,E1 18165.648,E2 18165.648} C_VEL
LIN {X 0,Y 402.984,Z 1094.295,A -85,B 0,C 180,E1 18163.717,E2 18163.717} C_VEL
LIN {X 0,Y 402.763,Z 1095.173,A -85,B 0,C 180,E1 18161.96,E2 18161.96} C_VEL
LIN {X 0,Y 402.675,Z 1094.8,A -85,B 0,C 180,E1 18160.414,E2 18160.414} C_VEL
LIN {X 0,Y 402.687,Z 1093.171,A -85,B 0,C 180,E1 18158.745,E2 18158.745} C_VEL
LIN {X 0,Y 402.844,Z 1089.936,A -85,B 0,C 180,E1 18156.91,E2 18156.91} C_VEL
LIN {X 0,Y 403.178,Z 1084.382,A -85,B 0,C 180,E1 18154.907,E2 18154.907} C_VEL
LIN {X 0,Y 403.574,Z 1078.544,A -85,B 0,C 180,E1 18153.356,E2 18153.356} C_VEL
LIN {X 0,Y 404.118,Z 1070.853,A -85,B 0,C 180,E1 18151.745,E2 18151.745} C_VEL
LIN {X 0,Y 404.818,Z 1060.604,A -85,B 0,C 180,E1 18150.07,E2 18150.07} C_VEL
LIN {X 0,Y 405.426,Z 1050.847,A -85,B 0,C 180,E1 18148.807,E2 18148.807} C_VEL
LIN {X 0,Y 406.01,Z 1040.351,A -85,B 0,C 180,E1 18147.696,E2 18147.696} C_VEL
LIN {X 0,Y 406.617,Z 1027.109,A -85,B 0,C 180,E1 18146.576,E2 18146.576} C_VEL
LIN {X 0,Y 407.042,Z 1013.702,A -85,B 0,C 180,E1 18145.732,E2 18145.732} C_VEL
LIN {X 0,Y 407.271,Z 1007.28,A -85,B 0,C 180,E1 18145.364,E2 18145.364} C_VEL
LIN {X 0,Y 408.339,Z 1007.772,A -85,B 0,C 180,E1 18145.041,E2 18145.041} C_VEL
LIN {X 0,Y 410.345,Z 1007.216,A -85,B 0,C 180,E1 18144.717,E2 18144.717} C_VEL
LIN {X 0,Y 413.331,Z 1005.406,A -85,B 0,C 180,E1 18144.423,E2 18144.423} C_VEL
LIN {X 0,Y 416.449,Z 1004.386,A -85,B 0,C 180,E1 18143.967,E2 18143.967} C_VEL
LIN {X 0,Y 420.682,Z 1001.951,A -85,B 0,C 180,E1 18143.544,E2 18143.544} C_VEL
LIN {X 0,Y 425.49,Z 999.583,A -85,B 0,C 180,E1 18143.016,E2 18143.016} C_VEL
LIN {X 0,Y 429.111,Z 997.281,A -85,B 0,C 180,E1 18142.711,E2 18142.711} C_VEL
LIN {X 0,Y 434.263,Z 994.325,A -85,B 0,C 180,E1 18142.232,E2 18142.232} C_VEL
LIN {X 0,Y 438.099,Z 991.701,A -85,B 0,C 180,E1 18141.958,E2 18141.958} C_VEL
LIN {X 0,Y 444.493,Z 987.656,A -85,B 0,C 180,E1 18141.456,E2 18141.456} C_VEL
LIN {X 0,Y 448.406,Z 984.882,A -85,B 0,C 180,E1 18141.2,E2 18141.2} C_VEL
LIN {X 0,Y 455.079,Z 980.187,A -85,B 0,C 180,E1 18140.744,E2 18140.744} C_VEL
LIN {X 0,Y 459.085,Z 977.072,A -85,B 0,C 180,E1 18140.507,E2 18140.507} C_VEL
LIN {X 0,Y 460.312,Z 976.325,A -85,B 0,C 180,E1 18140.411,E2 18140.411} C_VEL
LIN {X 0,Y 452.922,Z 1000.104,A -85,B 0,C 180,E1 18138.356,E2 18138.356} C_VEL
LIN {X 0,Y 446.484,Z 1019.668,A -85,B 0,C 180,E1 18136.389,E2 18136.389} C_VEL
LIN {X 0,Y 439.135,Z 1041.133,A -85,B 0,C 180,E1 18133.896,E2 18133.896} C_VEL
LIN {X 0,Y 433.243,Z 1057.866,A -85,B 0,C 180,E1 18131.659,E2 18131.659} C_VEL
LIN {X 0,Y 426.832,Z 1076.074,A -85,B 0,C 180,E1 18128.89,E2 18128.89} C_VEL
LIN {X 0,Y 421.171,Z 1092.055,A -85,B 0,C 180,E1 18126.071,E2 18126.071} C_VEL
LIN {X 0,Y 415.904,Z 1107.757,A -85,B 0,C 180,E1 18122.912,E2 18122.912} C_VEL
LIN {X 0,Y 411.46,Z 1121.294,A -85,B 0,C 180,E1 18119.72,E2 18119.72} C_VEL
LIN {X 0,Y 408.207,Z 1132.183,A -85,B 0,C 180,E1 18116.79,E2 18116.79} C_VEL
LIN {X 0,Y 405.041,Z 1143.941,A -85,B 0,C 180,E1 18113.112,E2 18113.112} C_VEL
LIN {X 0,Y 403.016,Z 1152.595,A -85,B 0,C 180,E1 18109.872,E2 18109.872} C_VEL
LIN {X 0,Y 401.662,Z 1159.579,A -85,B 0,C 180,E1 18106.786,E2 18106.786} C_VEL
LIN {X 0,Y 400.665,Z 1166.342,A -85,B 0,C 180,E1 18103.128,E2 18103.128} C_VEL
LIN {X 0,Y 400.199,Z 1170.936,A -85,B 0,C 180,E1 18099.783,E2 18099.783} C_VEL
LIN {X 0,Y 400.183,Z 1171.12,A -85,B 0,C 180,E1 18099.621,E2 18099.621} C_VEL
LIN {X 0,Y 399.101,Z 1172.419,A -85,B 0,C 180,E1 18098.534,E2 18098.534} C_VEL
LIN {X 0,Y 392.516,Z 1175.34,A -85,B 0,C 180,E1 18095.459,E2 18095.459} C_VEL
LIN {X 0,Y 391.961,Z 1175.77,A -85,B 0,C 180,E1 18094.65,E2 18094.65} C_VEL
LIN {X 0,Y 391.94,Z 1176.887,A -85,B 0,C 180,E1 18091.61,E2 18091.61} C_VEL
LIN {X 0,Y 391.94,Z 1176.973,A -85,B 0,C 180,E1 18088.832,E2 18088.832} C_VEL
LIN {X 0,Y 391.955,Z 1176.149,A -85,B 0,C 180,E1 18086.052,E2 18086.052} C_VEL
LIN {X 0,Y 392.015,Z 1174.416,A -85,B 0,C 180,E1 18083.264,E2 18083.264} C_VEL
LIN {X 0,Y 392.178,Z 1171.766,A -85,B 0,C 180,E1 18080.463,E2 18080.463} C_VEL
LIN {X 0,Y 392.553,Z 1167.971,A -85,B 0,C 180,E1 18077.498,E2 18077.498} C_VEL
LIN {X 0,Y 393.38,Z 1162.34,A -85,B 0,C 180,E1 18074.069,E2 18074.069} C_VEL
LIN {X 0,Y 394.907,Z 1154.448,A -85,B 0,C 180,E1 18070.323,E2 18070.323} C_VEL
LIN {X 0,Y 396.813,Z 1146.443,A -85,B 0,C 180,E1 18067.169,E2 18067.169} C_VEL
LIN {X 0,Y 399.515,Z 1136.681,A -85,B 0,C 180,E1 18063.868,E2 18063.868} C_VEL
LIN {X 0,Y 403.385,Z 1124.122,A -85,B 0,C 180,E1 18060.283,E2 18060.283} C_VEL
LIN {X 0,Y 407.383,Z 1112.126,A -85,B 0,C 180,E1 18057.321,E2 18057.321} C_VEL
LIN {X 0,Y 412.723,Z 1097.218,A -85,B 0,C 180,E1 18054.109,E2 18054.109} C_VEL
LIN {X 0,Y 418.484,Z 1081.289,A -85,B 0,C 180,E1 18051.162,E2 18051.162} C_VEL
LIN {X 0,Y 425.143,Z 1063.453,A -85,B 0,C 180,E1 18048.276,E2 18048.276} C_VEL
LIN {X 0,Y 431.83,Z 1045.088,A -85,B 0,C 180,E1 18045.727,E2 18045.727} C_VEL
LIN {X 0,Y 439.055,Z 1025.214,A -85,B 0,C 180,E1 18043.316,E2 18043.316} C_VEL
LIN {X 0,Y 446.158,Z 1004.37,A -85,B 0,C 180,E1 18041.151,E2 18041.151} C_VEL
LIN {X 0,Y 453.365,Z 982.514,A -85,B 0,C 180,E1 18039.178,E2 18039.178} C_VEL
LIN {X 0,Y 459.974,Z 960.546,A -85,B 0,C 180,E1 18037.493,E2 18037.493} C_VEL
LIN {X 0,Y 465.884,Z 939.59,A -85,B 0,C 180,E1 18036.098,E2 18036.098} C_VEL
LIN {X 0,Y 471.97,Z 915.203,A -85,B 0,C 180,E1 18034.719,E2 18034.719} C_VEL
LIN {X 0,Y 476.936,Z 893.107,A -85,B 0,C 180,E1 18033.668,E2 18033.668} C_VEL
LIN {X 0,Y 482.012,Z 866.564,A -85,B 0,C 180,E1 18032.63,E2 18032.63} C_VEL
LIN {X 0,Y 485.41,Z 845.118,A -85,B 0,C 180,E1 18031.951,E2 18031.951} C_VEL
LIN {X 0,Y 492.444,Z 796.283,A -85,B 0,C 180,E1 18030.727,E2 18030.727} C_VEL
LIN {X 0,Y 504.375,Z 709.08,A -85,B 0,C 180,E1 18028.799,E2 18028.799} C_VEL
LIN {X 0,Y 513.868,Z 631.384,A -85,B 0,C 180,E1 18027.266,E2 18027.266} C_VEL
LIN {X 0,Y 521.367,Z 558.159,A -85,B 0,C 180,E1 18025.962,E2 18025.962} C_VEL
LIN {X 0,Y 524.291,Z 522.66,A -85,B 0,C 180,E1 18025.35,E2 18025.35} C_VEL
LIN {X 0,Y 519.452,Z 518.461,A -85,B 0,C 180,E1 18024.024,E2 18024.024} C_VEL
LIN {X 0,Y 511.758,Z 512.303,A -85,B 0,C 180,E1 18021.731,E2 18021.731} C_VEL
LIN {X 0,Y 501.337,Z 505.068,A -85,B 0,C 180,E1 18018.128,E2 18018.128} C_VEL
LIN {X 0,Y 492.43,Z 501.144,A -85,B 0,C 180,E1 18014.343,E2 18014.343} C_VEL
LIN {X 0,Y 486.882,Z 499.43,A -85,B 0,C 180,E1 18011.251,E2 18011.251} C_VEL
LIN {X 0,Y 487.554,Z 500.477,A -85,B 0,C 180,E1 18009.086,E2 18009.086} C_VEL
LIN {X 0,Y 489.242,Z 504.773,A -85,B 0,C 180,E1 18005.042,E2 18005.042} C_VEL
LIN {X 0,Y 490.929,Z 508.983,A -85,B 0,C 180,E1 18002.335,E2 18002.335} C_VEL
LIN {X 0,Y 492.752,Z 513.476,A -85,B 0,C 180,E1 18000,E2 18000} C_VEL
LIN {X 0,Y 495.247,Z 519.597,A -85,B 0,C 180,E1 17997.338,E2 17997.338} C_VEL
LIN {X 0,Y 498.679,Z 528.684,A -85,B 0,C 180,E1 17994.131,E2 17994.131} C_VEL
LIN {X 0,Y 502.304,Z 538.629,A -85,B 0,C 180,E1 17991.183,E2 17991.183} C_VEL
LIN {X 0,Y 502.447,Z 539.047,A -85,B 0,C 180,E1 17991.07,E2 17991.07} C_VEL
LIN {X 0,Y 493.205,Z 570.161,A -85,B 0,C 180,E1 17988.131,E2 17988.131} C_VEL
LIN {X 0,Y 483.535,Z 604.807,A -85,B 0,C 180,E1 17984.94,E2 17984.94} C_VEL
LIN {X 0,Y 482.24,Z 610.539,A -85,B 0,C 180,E1 17984.447,E2 17984.447} C_VEL
LIN {X 0,Y 484.014,Z 649.87,A -85,B 0,C 180,E1 17981.824,E2 17981.824} C_VEL
LIN {X 0,Y 485.94,Z 671.768,A -85,B 0,C 180,E1 17980.215,E2 17980.215} C_VEL
LIN {X 0,Y 489.058,Z 694.545,A -85,B 0,C 180,E1 17978.344,E2 17978.344} C_VEL
LIN {X 0,Y 493.301,Z 715.728,A -85,B 0,C 180,E1 17976.368,E2 17976.368} C_VEL
LIN {X 0,Y 497.896,Z 733.215,A -85,B 0,C 180,E1 17974.563,E2 17974.563} C_VEL
LIN {X 0,Y 504.414,Z 752.155,A -85,B 0,C 180,E1 17972.412,E2 17972.412} C_VEL
LIN {X 0,Y 509.136,Z 763.083,A -85,B 0,C 180,E1 17971.059,E2 17971.059} C_VEL
LIN {X 0,Y 506.205,Z 783.812,A -85,B 0,C 180,E1 17970.798,E2 17970.798} C_VEL
LIN {X 0,Y 500.513,Z 823.972,A -85,B 0,C 180,E1 17969.945,E2 17969.945} C_VEL
LIN {X 0,Y 493.921,Z 861.128,A -85,B 0,C 180,E1 17969.014,E2 17969.014} C_VEL
LIN {X 0,Y 487.423,Z 893.882,A -85,B 0,C 180,E1 17967.962,E2 17967.962} C_VEL
LIN {X 0,Y 480.764,Z 925.114,A -85,B 0,C 180,E1 17966.724,E2 17966.724} C_VEL
LIN {X 0,Y 473.566,Z 956.555,A -85,B 0,C 180,E1 17965.215,E2 17965.215} C_VEL
LIN {X 0,Y 466.084,Z 987.317,A -85,B 0,C 180,E1 17963.454,E2 17963.454} C_VEL
LIN {X 0,Y 460.004,Z 1010.548,A -85,B 0,C 180,E1 17961.89,E2 17961.89} C_VEL
LIN {X 0,Y 453.676,Z 1032.047,A -85,B 0,C 180,E1 17960.179,E2 17960.179} C_VEL
LIN {X 0,Y 446.744,Z 1053.159,A -85,B 0,C 180,E1 17958.182,E2 17958.182} C_VEL
LIN {X 0,Y 439.972,Z 1072.039,A -85,B 0,C 180,E1 17956.086,E2 17956.086} C_VEL
LIN {X 0,Y 432.871,Z 1090.592,A -85,B 0,C 180,E1 17953.679,E2 17953.679} C_VEL
LIN {X 0,Y 425.978,Z 1107.654,A -85,B 0,C 180,E1 17951.087,E2 17951.087} C_VEL
LIN {X 0,Y 419.405,Z 1123.31,A -85,B 0,C 180,E1 17948.303,E2 17948.303} C_VEL
LIN {X 0,Y 413.001,Z 1138.189,A -85,B 0,C 180,E1 17945.181,E2 17945.181} C_VEL
LIN {X 0,Y 407.115,Z 1152.054,A -85,B 0,C 180,E1 17941.706,E2 17941.706} C_VEL
LIN {X 0,Y 402.287,Z 1163.79,A -85,B 0,C 180,E1 17938.178,E2 17938.178} C_VEL
LIN {X 0,Y 398.408,Z 1174.048,A -85,B 0,C 180,E1 17934.46,E2 17934.46} C_VEL
LIN {X 0,Y 395.494,Z 1182.821,A -85,B 0,C 180,E1 17930.572,E2 17930.572} C_VEL
LIN {X 0,Y 393.587,Z 1189.83,A -85,B 0,C 180,E1 17926.681,E2 17926.681} C_VEL
LIN {X 0,Y 392.522,Z 1195.234,A -85,B 0,C 180,E1 17922.802,E2 17922.802} C_VEL
LIN {X 0,Y 392.069,Z 1199.142,A -85,B 0,C 180,E1 17918.948,E2 17918.948} C_VEL
LIN {X 0,Y 391.946,Z 1201.564,A -85,B 0,C 180,E1 17915.268,E2 17915.268} C_VEL
LIN {X 0,Y 391.938,Z 1202.72,A -85,B 0,C 180,E1 17911.752,E2 17911.752} C_VEL
LIN {X 0,Y 391.939,Z 1202.72,A -85,B 0,C 180,E1 17908.244,E2 17908.244} C_VEL
LIN {X 0,Y 391.946,Z 1201.564,A -85,B 0,C 180,E1 17904.729,E2 17904.729} C_VEL
LIN {X 0,Y 392.068,Z 1199.141,A -85,B 0,C 180,E1 17901.049,E2 17901.049} C_VEL
LIN {X 0,Y 392.522,Z 1195.232,A -85,B 0,C 180,E1 17897.194,E2 17897.194} C_VEL
LIN {X 0,Y 393.601,Z 1189.769,A -85,B 0,C 180,E1 17893.28,E2 17893.28} C_VEL
LIN {X 0,Y 395.496,Z 1182.811,A -85,B 0,C 180,E1 17889.424,E2 17889.424} C_VEL
LIN {X 0,Y 398.412,Z 1174.037,A -85,B 0,C 180,E1 17885.536,E2 17885.536} C_VEL
LIN {X 0,Y 402.289,Z 1163.775,A -85,B 0,C 180,E1 17881.818,E2 17881.818} C_VEL
LIN {X 0,Y 407.118,Z 1152.031,A -85,B 0,C 180,E1 17878.291,E2 17878.291} C_VEL
LIN {X 0,Y 413.004,Z 1138.156,A -85,B 0,C 180,E1 17874.815,E2 17874.815} C_VEL
LIN {X 0,Y 419.53,Z 1123.006,A -85,B 0,C 180,E1 17871.64,E2 17871.64} C_VEL
LIN {X 0,Y 426.333,Z 1106.795,A -85,B 0,C 180,E1 17868.772,E2 17868.772} C_VEL
LIN {X 0,Y 433.385,Z 1089.259,A -85,B 0,C 180,E1 17866.134,E2 17866.134} C_VEL
LIN {X 0,Y 440.55,Z 1070.421,A -85,B 0,C 180,E1 17863.724,E2 17863.724} C_VEL
LIN {X 0,Y 447.612,Z 1050.472,A -85,B 0,C 180,E1 17861.552,E2 17861.552} C_VEL
LIN {X 0,Y 454.359,Z 1029.657,A -85,B 0,C 180,E1 17859.624,E2 17859.624} C_VEL
LIN {X 0,Y 460.757,Z 1007.822,A -85,B 0,C 180,E1 17857.912,E2 17857.912} C_VEL
LIN {X 0,Y 467.085,Z 983.17,A -85,B 0,C 180,E1 17856.294,E2 17856.294} C_VEL
LIN {X 0,Y 474.856,Z 951.069,A -85,B 0,C 180,E1 17854.502,E2 17854.502} C_VEL
LIN {X 0,Y 481.91,Z 919.615,A -85,B 0,C 180,E1 17853.044,E2 17853.044} C_VEL
LIN {X 0,Y 488.815,Z 886.816,A -85,B 0,C 180,E1 17851.796,E2 17851.796} C_VEL
LIN {X 0,Y 495.439,Z 852.746,A -85,B 0,C 180,E1 17850.763,E2 17850.763} C_VEL
LIN {X 0,Y 502.168,Z 812.982,A -85,B 0,C 180,E1 17849.812,E2 17849.812} C_VEL
LIN {X 0,Y 507.269,Z 773.74,A -85,B 0,C 180,E1 17849.015,E2 17849.015} C_VEL
LIN {X 0,Y 511.245,Z 732.69,A -85,B 0,C 180,E1 17848.336,E2 17848.336} C_VEL
LIN {X 0,Y 516.148,Z 666.708,A -85,B 0,C 180,E1 17847.461,E2 17847.461} C_VEL
LIN {X 0,Y 517.624,Z 650.639,A -85,B 0,C 180,E1 17847.205,E2 17847.205} C_VEL
LIN {X 0,Y 523.21,Z 610.685,A -85,B 0,C 180,E1 17846.6,E2 17846.6} C_VEL
LIN {X 0,Y 527.875,Z 575.078,A -85,B 0,C 180,E1 17846,E2 17846} C_VEL
LIN {X 0,Y 531.975,Z 547.261,A -85,B 0,C 180,E1 17845.623,E2 17845.623} C_VEL
LIN {X 0,Y 534.373,Z 528.199,A -85,B 0,C 180,E1 17845.281,E2 17845.281} C_VEL
LIN {X 0,Y 526.486,Z 514.24,A -85,B 0,C 180,E1 17842.904,E2 17842.904} C_VEL
LIN {X 0,Y 520.196,Z 528.47,A -85,B 0,C 180,E1 17842.107,E2 17842.107} C_VEL
LIN {X 0,Y 512.85,Z 546.662,A -85,B 0,C 180,E1 17841.203,E2 17841.203} C_VEL
LIN {X 0,Y 509.123,Z 555.288,A -85,B 0,C 180,E1 17840.687,E2 17840.687} C_VEL
LIN {X 0,Y 503.17,Z 570.688,A -85,B 0,C 180,E1 17839.917,E2 17839.917} C_VEL
LIN {X 0,Y 499.16,Z 580.29,A -85,B 0,C 180,E1 17839.328,E2 17839.328} C_VEL
LIN {X 0,Y 493.351,Z 595.984,A -85,B 0,C 180,E1 17838.539,E2 17838.539} C_VEL
LIN {X 0,Y 489.121,Z 606.47,A -85,B 0,C 180,E1 17837.872,E2 17837.872} C_VEL
LIN {X 0,Y 485.443,Z 618.591,A -85,B 0,C 180,E1 17837.3,E2 17837.3} C_VEL
LIN {X 0,Y 480.914,Z 634.75,A -85,B 0,C 180,E1 17836.348,E2 17836.348} C_VEL
LIN {X 0,Y 479.751,Z 639.271,A -85,B 0,C 180,E1 17836.11,E2 17836.11} C_VEL
LIN {X 0,Y 474.617,Z 661.054,A -85,B 0,C 180,E1 17835.097,E2 17835.097} C_VEL
LIN {X 0,Y 470.085,Z 678.192,A -85,B 0,C 180,E1 17834.074,E2 17834.074} C_VEL
LIN {X 0,Y 468.819,Z 682.878,A -85,B 0,C 180,E1 17833.804,E2 17833.804} C_VEL
LIN {X 0,Y 463.533,Z 703.43,A -85,B 0,C 180,E1 17832.809,E2 17832.809} C_VEL
LIN {X 0,Y 459.002,Z 718.307,A -85,B 0,C 180,E1 17831.848,E2 17831.848} C_VEL
LIN {X 0,Y 457.777,Z 722.35,A -85,B 0,C 180,E1 17831.601,E2 17831.601} C_VEL
LIN {X 0,Y 452.582,Z 740.187,A -85,B 0,C 180,E1 17830.671,E2 17830.671} C_VEL
LIN {X 0,Y 448.5,Z 752.376,A -85,B 0,C 180,E1 17829.799,E2 17829.799} C_VEL
LIN {X 0,Y 447.236,Z 756.325,A -85,B 0,C 180,E1 17829.558,E2 17829.558} C_VEL
LIN {X 0,Y 442.16,Z 772.27,A -85,B 0,C 180,E1 17828.649,E2 17828.649} C_VEL
LIN {X 0,Y 437.986,Z 784.06,A -85,B 0,C 180,E1 17827.741,E2 17827.741} C_VEL
LIN {X 0,Y 432.988,Z 799.08,A -85,B 0,C 180,E1 17826.846,E2 17826.846} C_VEL
LIN {X 0,Y 429.415,Z 808.79,A -85,B 0,C 180,E1 17826.015,E2 17826.015} C_VEL
LIN {X 0,Y 424.524,Z 823.233,A -85,B 0,C 180,E1 17825.127,E2 17825.127} C_VEL
LIN {X 0,Y 421.149,Z 832.461,A -85,B 0,C 180,E1 17824.307,E2 17824.307} C_VEL
LIN {X 0,Y 415.752,Z 848.052,A -85,B 0,C 180,E1 17823.257,E2 17823.257} C_VEL
LIN {X 0,Y 413.019,Z 855.344,A -85,B 0,C 180,E1 17822.515,E2 17822.515} C_VEL
LIN {X 0,Y 407.522,Z 871.306,A -85,B 0,C 180,E1 17821.547,E2 17821.547} C_VEL
LIN {X 0,Y 404.399,Z 880.105,A -85,B 0,C 180,E1 17820.779,E2 17820.779} C_VEL
LIN {X 0,Y 403.987,Z 881.583,A -85,B 0,C 180,E1 17820.641,E2 17820.641} C_VEL
LIN {X 0,Y 403.535,Z 887.725,A -85,B 0,C 180,E1 17820.426,E2 17820.426} C_VEL
LIN {X 0,Y 400.989,Z 981.142,A -85,B 0,C 180,E1 17818.312,E2 17818.312} C_VEL
LIN {X 0,Y 401.05,Z 1002.749,A -85,B 0,C 180,E1 17817.75,E2 17817.75} C_VEL
LIN {X 0,Y 400.936,Z 1017.415,A -85,B 0,C 180,E1 17817.141,E2 17817.141} C_VEL
LIN {X 0,Y 400.538,Z 1030.438,A -85,B 0,C 180,E1 17816.35,E2 17816.35} C_VEL
LIN {X 0,Y 400.067,Z 1041.488,A -85,B 0,C 180,E1 17815.485,E2 17815.485} C_VEL
LIN {X 0,Y 399.405,Z 1053.194,A -85,B 0,C 180,E1 17814.331,E2 17814.331} C_VEL
LIN {X 0,Y 398.565,Z 1063.993,A -85,B 0,C 180,E1 17812.939,E2 17812.939} C_VEL
LIN {X 0,Y 397.91,Z 1071.353,A -85,B 0,C 180,E1 17811.765,E2 17811.765} C_VEL
LIN {X 0,Y 397.234,Z 1078.145,A -85,B 0,C 180,E1 17810.437,E2 17810.437} C_VEL
LIN {X 0,Y 396.572,Z 1084.222,A -85,B 0,C 180,E1 17808.953,E2 17808.953} C_VEL
LIN {X 0,Y 395.925,Z 1089.792,A -85,B 0,C 180,E1 17807.159,E2 17807.159} C_VEL
LIN {X 0,Y 395.369,Z 1093.729,A -85,B 0,C 180,E1 17805.201,E2 17805.201} C_VEL
LIN {X 0,Y 395.039,Z 1095.653,A -85,B 0,C 180,E1 17803.532,E2 17803.532} C_VEL
LIN {X 0,Y 394.849,Z 1096.316,A -85,B 0,C 180,E1 17802.004,E2 17802.004} C_VEL
LIN {X 0,Y 394.749,Z 1095.84,A -85,B 0,C 180,E1 17800.313,E2 17800.313} C_VEL
LIN {X 0,Y 394.767,Z 1094.1,A -85,B 0,C 180,E1 17798.609,E2 17798.609} C_VEL
LIN {X 0,Y 394.963,Z 1090.374,A -85,B 0,C 180,E1 17796.58,E2 17796.58} C_VEL
LIN {X 0,Y 395.29,Z 1084.948,A -85,B 0,C 180,E1 17794.692,E2 17794.692} C_VEL
LIN {X 0,Y 395.713,Z 1078.956,A -85,B 0,C 180,E1 17793.109,E2 17793.109} C_VEL
LIN {X 0,Y 396.339,Z 1070.543,A -85,B 0,C 180,E1 17791.358,E2 17791.358} C_VEL
LIN {X 0,Y 397.025,Z 1060.456,A -85,B 0,C 180,E1 17789.751,E2 17789.751} C_VEL
LIN {X 0,Y 397.666,Z 1050.454,A -85,B 0,C 180,E1 17788.466,E2 17788.466} C_VEL
LIN {X 0,Y 398.374,Z 1037.942,A -85,B 0,C 180,E1 17787.17,E2 17787.17} C_VEL
LIN {X 0,Y 398.926,Z 1024.903,A -85,B 0,C 180,E1 17786.142,E2 17786.142} C_VEL
LIN {X 0,Y 399.25,Z 1015.282,A -85,B 0,C 180,E1 17785.528,E2 17785.528} C_VEL
LIN {X 0,Y 400.546,Z 1015.792,A -85,B 0,C 180,E1 17785.134,E2 17785.134} C_VEL
LIN {X 0,Y 402.558,Z 1015.211,A -85,B 0,C 180,E1 17784.813,E2 17784.813} C_VEL
LIN {X 0,Y 404.938,Z 1014.067,A -85,B 0,C 180,E1 17784.53,E2 17784.53} C_VEL
LIN {X 0,Y 408.335,Z 1013.064,A -85,B 0,C 180,E1 17784.007,E2 17784.007} C_VEL
LIN {X 0,Y 411.646,Z 1011.333,A -85,B 0,C 180,E1 17783.653,E2 17783.653} C_VEL
LIN {X 0,Y 416.222,Z 1009.464,A -85,B 0,C 180,E1 17783.089,E2 17783.089} C_VEL
LIN {X 0,Y 419.658,Z 1007.615,A -85,B 0,C 180,E1 17782.757,E2 17782.757} C_VEL
LIN {X 0,Y 425.542,Z 1004.611,A -85,B 0,C 180,E1 17782.174,E2 17782.174} C_VEL
LIN {X 0,Y 429.15,Z 1002.517,A -85,B 0,C 180,E1 17781.871,E2 17781.871} C_VEL
LIN {X 0,Y 435.442,Z 998.785,A -85,B 0,C 180,E1 17781.348,E2 17781.348} C_VEL
LIN {X 0,Y 439.188,Z 996.386,A -85,B 0,C 180,E1 17781.07,E2 17781.07} C_VEL
LIN {X 0,Y 445.822,Z 992.012,A -85,B 0,C 180,E1 17780.601,E2 17780.601} C_VEL
LIN {X 0,Y 451.387,Z 988.344,A -85,B 0,C 180,E1 17780.226,E2 17780.226} C_VEL
LIN {X 0,Y 444.818,Z 1008.319,A -85,B 0,C 180,E1 17778.368,E2 17778.368} C_VEL
LIN {X 0,Y 437.096,Z 1030.39,A -85,B 0,C 180,E1 17775.99,E2 17775.99} C_VEL
LIN {X 0,Y 430.313,Z 1049.208,A -85,B 0,C 180,E1 17773.641,E2 17773.641} C_VEL
LIN {X 0,Y 423.264,Z 1068.33,A -85,B 0,C 180,E1 17770.873,E2 17770.873} C_VEL
LIN {X 0,Y 417.322,Z 1084.496,A -85,B 0,C 180,E1 17768.183,E2 17768.183} C_VEL
LIN {X 0,Y 411.037,Z 1101.722,A -85,B 0,C 180,E1 17764.868,E2 17764.868} C_VEL
LIN {X 0,Y 406.418,Z 1114.964,A -85,B 0,C 180,E1 17761.92,E2 17761.92} C_VEL
LIN {X 0,Y 401.732,Z 1129.266,A -85,B 0,C 180,E1 17758.224,E2 17758.224} C_VEL
LIN {X 0,Y 398.636,Z 1139.633,A -85,B 0,C 180,E1 17755.083,E2 17755.083} C_VEL
LIN {X 0,Y 396.072,Z 1149.477,A -85,B 0,C 180,E1 17751.63,E2 17751.63} C_VEL
LIN {X 0,Y 394.116,Z 1158.23,A -85,B 0,C 180,E1 17747.879,E2 17747.879} C_VEL
LIN {X 0,Y 393.085,Z 1164.066,A -85,B 0,C 180,E1 17744.848,E2 17744.848} C_VEL
LIN {X 0,Y 392.463,Z 1168.683,A -85,B 0,C 180,E1 17741.911,E2 17741.911} C_VEL
LIN {X 0,Y 392.137,Z 1172.482,A -85,B 0,C 180,E1 17738.802,E2 17738.802} C_VEL
LIN {X 0,Y 391.976,Z 1175.545,A -85,B 0,C 180,E1 17735.124,E2 17735.124} C_VEL
LIN {X 0,Y 391.961,Z 1175.77,A -85,B 0,C 180,E1 17734.65,E2 17734.65} C_VEL
LIN {X 0,Y 390.949,Z 1176.35,A -85,B 0,C 180,E1 17733.527,E2 17733.527} C_VEL
LIN {X 0,Y 386.667,Z 1177.167,A -85,B 0,C 180,E1 17731.564,E2 17731.564} C_VEL
LIN {X 0,Y 384.145,Z 1177.402,A -85,B 0,C 180,E1 17730.025,E2 17730.025} C_VEL
LIN {X 0,Y 383.938,Z 1177.349,A -85,B 0,C 180,E1 17729.525,E2 17729.525} C_VEL
LIN {X 0,Y 383.959,Z 1176.547,A -85,B 0,C 180,E1 17726.269,E2 17726.269} C_VEL
LIN {X 0,Y 384.022,Z 1174.783,A -85,B 0,C 180,E1 17723.273,E2 17723.273} C_VEL
LIN {X 0,Y 384.193,Z 1172.172,A -85,B 0,C 180,E1 17720.414,E2 17720.414} C_VEL
LIN {X 0,Y 384.588,Z 1168.415,A -85,B 0,C 180,E1 17717.388,E2 17717.388} C_VEL
LIN {X 0,Y 385.357,Z 1163.346,A -85,B 0,C 180,E1 17714.192,E2 17714.192} C_VEL
LIN {X 0,Y 387.044,Z 1155.124,A -85,B 0,C 180,E1 17710.113,E2 17710.113} C_VEL
LIN {X 0,Y 389.068,Z 1147.06,A -85,B 0,C 180,E1 17706.848,E2 17706.848} C_VEL
LIN {X 0,Y 391.907,Z 1137.359,A -85,B 0,C 180,E1 17703.484,E2 17703.484} C_VEL
LIN {X 0,Y 395.955,Z 1124.892,A -85,B 0,C 180,E1 17699.835,E2 17699.835} C_VEL
LIN {X 0,Y 400.142,Z 1112.969,A -85,B 0,C 180,E1 17696.824,E2 17696.824} C_VEL
LIN {X 0,Y 405.699,Z 1098.164,A -85,B 0,C 180,E1 17693.564,E2 17693.564} C_VEL
LIN {X 0,Y 411.737,Z 1082.215,A -85,B 0,C 180,E1 17690.557,E2 17690.557} C_VEL
LIN {X 0,Y 418.603,Z 1064.615,A -85,B 0,C 180,E1 17687.658,E2 17687.658} C_VEL
LIN {X 0,Y 425.525,Z 1046.361,A -85,B 0,C 180,E1 17685.084,E2 17685.084} C_VEL
LIN {X 0,Y 432.985,Z 1026.625,A -85,B 0,C 180,E1 17682.653,E2 17682.653} C_VEL
LIN {X 0,Y 440.308,Z 1005.921,A -85,B 0,C 180,E1 17680.473,E2 17680.473} C_VEL
LIN {X 0,Y 447.482,Z 984.982,A -85,B 0,C 180,E1 17678.553,E2 17678.553} C_VEL
LIN {X 0,Y 454.255,Z 963.303,A -85,B 0,C 180,E1 17676.862,E2 17676.862} C_VEL
LIN {X 0,Y 459.767,Z 944.478,A -85,B 0,C 180,E1 17675.578,E2 17675.578} C_VEL
LIN {X 0,Y 466.555,Z 918.738,A -85,B 0,C 180,E1 17674.077,E2 17674.077} C_VEL
LIN {X 0,Y 471.483,Z 897.524,A -85,B 0,C 180,E1 17673.046,E2 17673.046} C_VEL
LIN {X 0,Y 476.537,Z 872.897,A -85,B 0,C 180,E1 17672.036,E2 17672.036} C_VEL
LIN {X 0,Y 480.53,Z 849.041,A -85,B 0,C 180,E1 17671.257,E2 17671.257} C_VEL
LIN {X 0,Y 486.588,Z 808.162,A -85,B 0,C 180,E1 17670.197,E2 17670.197} C_VEL
LIN {X 0,Y 498.655,Z 724.002,A -85,B 0,C 180,E1 17668.299,E2 17668.299} C_VEL
LIN {X 0,Y 508.521,Z 647.057,A -85,B 0,C 180,E1 17666.751,E2 17666.751} C_VEL
LIN {X 0,Y 516.336,Z 575.532,A -85,B 0,C 180,E1 17665.454,E2 17665.454} C_VEL
LIN {X 0,Y 520.55,Z 528.582,A -85,B 0,C 180,E1 17664.661,E2 17664.661} C_VEL
LIN {X 0,Y 515.412,Z 524.297,A -85,B 0,C 180,E1 17663.192,E2 17663.192} C_VEL
LIN {X 0,Y 509.965,Z 519.89,A -85,B 0,C 180,E1 17661.509,E2 17661.509} C_VEL
LIN {X 0,Y 500.102,Z 512.946,A -85,B 0,C 180,E1 17658.053,E2 17658.053} C_VEL
LIN {X 0,Y 491.479,Z 509.092,A -85,B 0,C 180,E1 17654.371,E2 17654.371} C_VEL
LIN {X 0,Y 485.052,Z 507.328,A -85,B 0,C 180,E1 17650.812,E2 17650.812} C_VEL
LIN {X 0,Y 483.297,Z 506.868,A -85,B 0,C 180,E1 17649.527,E2 17649.527} C_VEL
LIN {X 0,Y 484.926,Z 511.37,A -85,B 0,C 180,E1 17645.205,E2 17645.205} C_VEL
LIN {X 0,Y 486.623,Z 515.803,A -85,B 0,C 180,E1 17642.355,E2 17642.355} C_VEL
LIN {X 0,Y 488.333,Z 520.072,A -85,B 0,C 180,E1 17640.117,E2 17640.117} C_VEL
LIN {X 0,Y 490.868,Z 526.538,A -85,B 0,C 180,E1 17637.315,E2 17637.315} C_VEL
LIN {X 0,Y 494.149,Z 535.334,A -85,B 0,C 180,E1 17634.193,E2 17634.193} C_VEL
LIN {X 0,Y 497.276,Z 544.282,A -85,B 0,C 180,E1 17631.53,E2 17631.53} C_VEL
LIN {X 0,Y 487.384,Z 576.701,A -85,B 0,C 180,E1 17628.461,E2 17628.461} C_VEL
LIN {X 0,Y 479.689,Z 604.199,A -85,B 0,C 180,E1 17625.938,E2 17625.938} C_VEL
LIN {X 0,Y 481.685,Z 658.596,A -85,B 0,C 180,E1 17622.264,E2 17622.264} C_VEL
LIN {X 0,Y 484.022,Z 683.72,A -85,B 0,C 180,E1 17620.34,E2 17620.34} C_VEL
LIN {X 0,Y 487.141,Z 705.186,A -85,B 0,C 180,E1 17618.476,E2 17618.476} C_VEL
LIN {X 0,Y 490.473,Z 722.308,A -85,B 0,C 180,E1 17616.83,E2 17616.83} C_VEL
LIN {X 0,Y 494.607,Z 738.7,A -85,B 0,C 180,E1 17615.118,E2 17615.118} C_VEL
LIN {X 0,Y 501,Z 757.986,A -85,B 0,C 180,E1 17612.9,E2 17612.9} C_VEL
LIN {X 0,Y 504.589,Z 766.659,A -85,B 0,C 180,E1 17611.814,E2 17611.814} C_VEL
LIN {X 0,Y 501.605,Z 787.354,A -85,B 0,C 180,E1 17611.512,E2 17611.512} C_VEL
LIN {X 0,Y 495.669,Z 827.4,A -85,B 0,C 180,E1 17610.647,E2 17610.647} C_VEL
LIN {X 0,Y 488.697,Z 864.708,A -85,B 0,C 180,E1 17609.683,E2 17609.683} C_VEL
LIN {X 0,Y 481.896,Z 897.832,A -85,B 0,C 180,E1 17608.592,E2 17608.592} C_VEL
LIN {X 0,Y 475.066,Z 928.768,A -85,B 0,C 180,E1 17607.337,E2 17607.337} C_VEL
LIN {X 0,Y 468.022,Z 958.781,A -85,B 0,C 180,E1 17605.876,E2 17605.876} C_VEL
LIN {X 0,Y 460.613,Z 988.254,A -85,B 0,C 180,E1 17604.169,E2 17604.169} C_VEL
LIN {X 0,Y 454.551,Z 1010.501,A -85,B 0,C 180,E1 17602.656,E2 17602.656} C_VEL
LIN {X 0,Y 448.38,Z 1030.84,A -85,B 0,C 180,E1 17601.034,E2 17601.034} C_VEL
LIN {X 0,Y 441.352,Z 1051.713,A -85,B 0,C 180,E1 17599.07,E2 17599.07} C_VEL
LIN {X 0,Y 434.254,Z 1070.912,A -85,B 0,C 180,E1 17596.939,E2 17596.939} C_VEL
LIN {X 0,Y 426.942,Z 1089.403,A -85,B 0,C 180,E1 17594.538,E2 17594.538} C_VEL
LIN {X 0,Y 419.599,Z 1107.006,A -85,B 0,C 180,E1 17591.851,E2 17591.851} C_VEL
LIN {X 0,Y 412.773,Z 1122.72,A -85,B 0,C 180,E1 17589.034,E2 17589.034} C_VEL
LIN {X 0,Y 406.115,Z 1137.679,A -85,B 0,C 180,E1 17585.869,E2 17585.869} C_VEL
LIN {X 0,Y 399.96,Z 1151.619,A -85,B 0,C 180,E1 17582.341,E2 17582.341} C_VEL
LIN {X 0,Y 394.711,Z 1163.875,A -85,B 0,C 180,E1 17578.603,E2 17578.603} C_VEL
LIN {X 0,Y 390.519,Z 1174.538,A -85,B 0,C 180,E1 17574.639,E2 17574.639} C_VEL
LIN {X 0,Y 387.454,Z 1183.437,A -85,B 0,C 180,E1 17570.544,E2 17570.544} C_VEL
LIN {X 0,Y 385.492,Z 1190.514,A -85,B 0,C 180,E1 17566.421,E2 17566.421} C_VEL
LIN {X 0,Y 384.462,Z 1195.706,A -85,B 0,C 180,E1 17562.464,E2 17562.464} C_VEL
LIN {X 0,Y 384.053,Z 1199.257,A -85,B 0,C 180,E1 17558.683,E2 17558.683} C_VEL
LIN {X 0,Y 383.944,Z 1201.507,A -85,B 0,C 180,E1 17554.928,E2 17554.928} C_VEL
LIN {X 0,Y 383.948,Z 1202.498,A -85,B 0,C 180,E1 17551.341,E2 17551.341} C_VEL
LIN {X 0,Y 383.942,Z 1202.385,A -85,B 0,C 180,E1 17547.759,E2 17547.759} C_VEL
LIN {X 0,Y 383.956,Z 1201.089,A -85,B 0,C 180,E1 17544.156,E2 17544.156} C_VEL
LIN {X 0,Y 384.114,Z 1198.504,A -85,B 0,C 180,E1 17540.408,E2 17540.408} C_VEL
LIN {X 0,Y 384.677,Z 1194.382,A -85,B 0,C 180,E1 17536.444,E2 17536.444} C_VEL
LIN {X 0,Y 385.959,Z 1188.558,A -85,B 0,C 180,E1 17532.354,E2 17532.354} C_VEL
LIN {X 0,Y 388.236,Z 1180.935,A -85,B 0,C 180,E1 17528.229,E2 17528.229} C_VEL
LIN {X 0,Y 391.535,Z 1171.759,A -85,B 0,C 180,E1 17524.268,E2 17524.268} C_VEL
LIN {X 0,Y 395.862,Z 1161.052,A -85,B 0,C 180,E1 17520.491,E2 17520.491} C_VEL
LIN {X 0,Y 401.207,Z 1148.643,A -85,B 0,C 180,E1 17516.865,E2 17516.865} C_VEL
LIN {X 0,Y 407.276,Z 1135.056,A -85,B 0,C 180,E1 17513.548,E2 17513.548} C_VEL
LIN {X 0,Y 413.746,Z 1120.477,A -85,B 0,C 180,E1 17510.535,E2 17510.535} C_VEL
LIN {X 0,Y 420.966,Z 1103.815,A -85,B 0,C 180,E1 17507.621,E2 17507.621} C_VEL
LIN {X 0,Y 428.342,Z 1085.957,A -85,B 0,C 180,E1 17504.983,E2 17504.983} C_VEL
LIN {X 0,Y 435.731,Z 1067.012,A -85,B 0,C 180,E1 17502.606,E2 17502.606} C_VEL
LIN {X 0,Y 443.177,Z 1046.351,A -85,B 0,C 180,E1 17500.405,E2 17500.405} C_VEL
LIN {X 0,Y 450.242,Z 1024.823,A -85,B 0,C 180,E1 17498.468,E2 17498.468} C_VEL
LIN {X 0,Y 456.534,Z 1003.564,A -85,B 0,C 180,E1 17496.847,E2 17496.847} C_VEL
LIN {X 0,Y 463.131,Z 978.231,A -85,B 0,C 180,E1 17495.228,E2 17495.228} C_VEL
LIN {X 0,Y 471.065,Z 945.854,A -85,B 0,C 180,E1 17493.467,E2 17493.467} C_VEL
LIN {X 0,Y 478.477,Z 913.45,A -85,B 0,C 180,E1 17492.014,E2 17492.014} C_VEL
LIN {X 0,Y 485.639,Z 879.761,A -85,B 0,C 180,E1 17490.785,E2 17490.785} C_VEL
LIN {X 0,Y 492.244,Z 846.002,A -85,B 0,C 180,E1 17489.811,E2 17489.811} C_VEL
LIN {X 0,Y 498.963,Z 806.103,A -85,B 0,C 180,E1 17488.881,E2 17488.881} C_VEL
LIN {X 0,Y 504.446,Z 763.209,A -85,B 0,C 180,E1 17488.041,E2 17488.041} C_VEL
LIN {X 0,Y 508.344,Z 721.278,A -85,B 0,C 180,E1 17487.386,E2 17487.386} C_VEL
LIN {X 0,Y 512.462,Z 666.888,A -85,B 0,C 180,E1 17486.67,E2 17486.67} C_VEL
LIN {X 0,Y 514.123,Z 647.713,A -85,B 0,C 180,E1 17486.374,E2 17486.374} C_VEL
LIN {X 0,Y 520.089,Z 605.041,A -85,B 0,C 180,E1 17485.716,E2 17485.716} C_VEL
LIN {X 0,Y 525.077,Z 568.832,A -85,B 0,C 180,E1 17485.143,E2 17485.143} C_VEL
LIN {X 0,Y 528.228,Z 547.701,A -85,B 0,C 180,E1 17484.86,E2 17484.86} C_VEL
LIN {X 0,Y 530.101,Z 532.615,A -85,B 0,C 180,E1 17484.577,E2 17484.577} C_VEL
LIN {X 0,Y 525.79,Z 525.106,A -85,B 0,C 180,E1 17483.268,E2 17483.268} C_VEL
LIN {X 0,Y 521.168,Z 535.407,A -85,B 0,C 180,E1 17482.69,E2 17482.69} C_VEL
LIN {X 0,Y 514.813,Z 550.92,A -85,B 0,C 180,E1 17481.925,E2 17481.925} C_VEL
LIN {X 0,Y 511.1,Z 559.424,A -85,B 0,C 180,E1 17481.429,E2 17481.429} C_VEL
LIN {X 0,Y 504.951,Z 575.036,A -85,B 0,C 180,E1 17480.654,E2 17480.654} C_VEL
LIN {X 0,Y 500.995,Z 584.4,A -85,B 0,C 180,E1 17480.092,E2 17480.092} C_VEL
LIN {X 0,Y 494.972,Z 600.349,A -85,B 0,C 180,E1 17479.294,E2 17479.294} C_VEL
LIN {X 0,Y 490.811,Z 610.522,A -85,B 0,C 180,E1 17478.661,E2 17478.661} C_VEL
LIN {X 0,Y 487.104,Z 622.626,A -85,B 0,C 180,E1 17478.093,E2 17478.093} C_VEL
LIN {X 0,Y 482.38,Z 639.037,A -85,B 0,C 180,E1 17477.132,E2 17477.132} C_VEL
LIN {X 0,Y 475.614,Z 666.72,A -85,B 0,C 180,E1 17475.83,E2 17475.83} C_VEL
LIN {X 0,Y 470.935,Z 683.581,A -85,B 0,C 180,E1 17474.808,E2 17474.808} C_VEL
LIN {X 0,Y 464.619,Z 707.473,A -85,B 0,C 180,E1 17473.654,E2 17473.654} C_VEL
LIN {X 0,Y 459.811,Z 722.753,A -85,B 0,C 180,E1 17472.671,E2 17472.671} C_VEL
LIN {X 0,Y 457.765,Z 729.774,A -85,B 0,C 180,E1 17472.312,E2 17472.312} C_VEL
LIN {X 0,Y 452.384,Z 747.12,A -85,B 0,C 180,E1 17471.361,E2 17471.361} C_VEL
LIN {X 0,Y 448.265,Z 759.016,A -85,B 0,C 180,E1 17470.515,E2 17470.515} C_VEL
LIN {X 0,Y 442.901,Z 775.434,A -85,B 0,C 180,E1 17469.601,E2 17469.601} C_VEL
LIN {X 0,Y 438.341,Z 788.012,A -85,B 0,C 180,E1 17468.659,E2 17468.659} C_VEL
LIN {X 0,Y 433.113,Z 803.222,A -85,B 0,C 180,E1 17467.753,E2 17467.753} C_VEL
LIN {X 0,Y 428.953,Z 814.26,A -85,B 0,C 180,E1 17466.866,E2 17466.866} C_VEL
LIN {X 0,Y 424.152,Z 827.812,A -85,B 0,C 180,E1 17466.019,E2 17466.019} C_VEL
LIN {X 0,Y 420.177,Z 838.357,A -85,B 0,C 180,E1 17465.12,E2 17465.12} C_VEL
LIN {X 0,Y 415.571,Z 851.214,A -85,B 0,C 180,E1 17464.278,E2 17464.278} C_VEL
LIN {X 0,Y 412.012,Z 860.627,A -85,B 0,C 180,E1 17463.417,E2 17463.417} C_VEL
LIN {X 0,Y 406.843,Z 875.079,A -85,B 0,C 180,E1 17462.536,E2 17462.536} C_VEL
LIN {X 0,Y 403.358,Z 884.616,A -85,B 0,C 180,E1 17461.705,E2 17461.705} C_VEL
LIN {X 0,Y 398.34,Z 898.737,A -85,B 0,C 180,E1 17461.098,E2 17461.098} C_VEL
LIN {X 0,Y 395.984,Z 905.205,A -85,B 0,C 180,E1 17460.598,E2 17460.598} C_VEL
LIN {X 0,Y 395.581,Z 906.719,A -85,B 0,C 180,E1 17460.462,E2 17460.462} C_VEL
LIN {X 0,Y 393.533,Z 983.466,A -85,B 0,C 180,E1 17458.685,E2 17458.685} C_VEL
LIN {X 0,Y 393.566,Z 1004.388,A -85,B 0,C 180,E1 17458.112,E2 17458.112} C_VEL
LIN {X 0,Y 393.389,Z 1019.486,A -85,B 0,C 180,E1 17457.451,E2 17457.451} C_VEL
LIN {X 0,Y 392.95,Z 1032.243,A -85,B 0,C 180,E1 17456.645,E2 17456.645} C_VEL
LIN {X 0,Y 392.451,Z 1043.194,A -85,B 0,C 180,E1 17455.763,E2 17455.763} C_VEL
LIN {X 0,Y 391.729,Z 1055.076,A -85,B 0,C 180,E1 17454.557,E2 17454.557} C_VEL
LIN {X 0,Y 390.861,Z 1065.525,A -85,B 0,C 180,E1 17453.168,E2 17453.168} C_VEL
LIN {X 0,Y 390.131,Z 1073.253,A -85,B 0,C 180,E1 17451.896,E2 17451.896} C_VEL
LIN {X 0,Y 389.425,Z 1079.935,A -85,B 0,C 180,E1 17450.542,E2 17450.542} C_VEL
LIN {X 0,Y 388.729,Z 1085.876,A -85,B 0,C 180,E1 17449.027,E2 17449.027} C_VEL
LIN {X 0,Y 387.99,Z 1091.629,A -85,B 0,C 180,E1 17447.044,E2 17447.044} C_VEL
LIN {X 0,Y 387.462,Z 1095.07,A -85,B 0,C 180,E1 17445.198,E2 17445.198} C_VEL
LIN {X 0,Y 387.146,Z 1096.79,A -85,B 0,C 180,E1 17443.649,E2 17443.649} C_VEL
LIN {X 0,Y 386.928,Z 1097.46,A -85,B 0,C 180,E1 17441.988,E2 17441.988} C_VEL
LIN {X 0,Y 386.826,Z 1096.976,A -85,B 0,C 180,E1 17440.365,E2 17440.365} C_VEL
LIN {X 0,Y 386.837,Z 1095.222,A -85,B 0,C 180,E1 17438.626,E2 17438.626} C_VEL
LIN {X 0,Y 387.038,Z 1091.357,A -85,B 0,C 180,E1 17436.511,E2 17436.511} C_VEL
LIN {X 0,Y 387.372,Z 1085.977,A -85,B 0,C 180,E1 17434.614,E2 17434.614} C_VEL
LIN {X 0,Y 387.805,Z 1080.014,A -85,B 0,C 180,E1 17433.013,E2 17433.013} C_VEL
LIN {X 0,Y 388.453,Z 1071.58,A -85,B 0,C 180,E1 17431.227,E2 17431.227} C_VEL
LIN {X 0,Y 389.16,Z 1061.485,A -85,B 0,C 180,E1 17429.591,E2 17429.591} C_VEL
LIN {X 0,Y 389.759,Z 1052.459,A -85,B 0,C 180,E1 17428.401,E2 17428.401} C_VEL
LIN {X 0,Y 390.366,Z 1042.212,A -85,B 0,C 180,E1 17427.285,E2 17427.285} C_VEL
LIN {X 0,Y 391.015,Z 1028.82,A -85,B 0,C 180,E1 17426.119,E2 17426.119} C_VEL
LIN {X 0,Y 391.272,Z 1023.133,A -85,B 0,C 180,E1 17425.703,E2 17425.703} C_VEL
LIN {X 0,Y 392.862,Z 1023.572,A -85,B 0,C 180,E1 17425.242,E2 17425.242} C_VEL
LIN {X 0,Y 395.737,Z 1022.496,A -85,B 0,C 180,E1 17424.825,E2 17424.825} C_VEL
LIN {X 0,Y 396.531,Z 1022.112,A -85,B 0,C 180,E1 17424.729,E2 17424.729} C_VEL
LIN {X 0,Y 399.8,Z 1021.329,A -85,B 0,C 180,E1 17424.181,E2 17424.181} C_VEL
LIN {X 0,Y 402.82,Z 1020.098,A -85,B 0,C 180,E1 17423.788,E2 17423.788} C_VEL
LIN {X 0,Y 407.224,Z 1018.512,A -85,B 0,C 180,E1 17423.193,E2 17423.193} C_VEL
LIN {X 0,Y 410.453,Z 1016.997,A -85,B 0,C 180,E1 17422.833,E2 17422.833} C_VEL
LIN {X 0,Y 416.462,Z 1014.259,A -85,B 0,C 180,E1 17422.178,E2 17422.178} C_VEL
LIN {X 0,Y 424.958,Z 1009.906,A -85,B 0,C 180,E1 17421.369,E2 17421.369} C_VEL
LIN {X 0,Y 435.671,Z 1003.77,A -85,B 0,C 180,E1 17420.526,E2 17420.526} C_VEL
LIN {X 0,Y 442.439,Z 999.767,A -85,B 0,C 180,E1 17420.034,E2 17420.034} C_VEL
LIN {X 0,Y 435.082,Z 1020.465,A -85,B 0,C 180,E1 17417.93,E2 17417.93} C_VEL
LIN {X 0,Y 427.523,Z 1041.111,A -85,B 0,C 180,E1 17415.508,E2 17415.508} C_VEL
LIN {X 0,Y 420.576,Z 1059.27,A -85,B 0,C 180,E1 17413.027,E2 17413.027} C_VEL
LIN {X 0,Y 413.636,Z 1077.402,A -85,B 0,C 180,E1 17410.193,E2 17410.193} C_VEL
LIN {X 0,Y 407.486,Z 1093.229,A -85,B 0,C 180,E1 17407.309,E2 17407.309} C_VEL
LIN {X 0,Y 401.956,Z 1108.126,A -85,B 0,C 180,E1 17404.209,E2 17404.209} C_VEL
LIN {X 0,Y 396.832,Z 1122.273,A -85,B 0,C 180,E1 17400.765,E2 17400.765} C_VEL
LIN {X 0,Y 393.079,Z 1133.599,A -85,B 0,C 180,E1 17397.58,E2 17397.58} C_VEL
LIN {X 0,Y 389.438,Z 1145.71,A -85,B 0,C 180,E1 17393.564,E2 17393.564} C_VEL
LIN {X 0,Y 387.356,Z 1153.722,A -85,B 0,C 180,E1 17390.396,E2 17390.396} C_VEL
LIN {X 0,Y 385.785,Z 1161.017,A -85,B 0,C 180,E1 17386.983,E2 17386.983} C_VEL
LIN {X 0,Y 384.684,Z 1167.649,A -85,B 0,C 180,E1 17383.071,E2 17383.071} C_VEL
LIN {X 0,Y 384.232,Z 1171.742,A -85,B 0,C 180,E1 17379.891,E2 17379.891} C_VEL
LIN {X 0,Y 384.036,Z 1174.477,A -85,B 0,C 180,E1 17377.031,E2 17377.031} C_VEL
LIN {X 0,Y 383.96,Z 1176.315,A -85,B 0,C 180,E1 17374.136,E2 17374.136} C_VEL
LIN {X 0,Y 383.945,Z 1177.197,A -85,B 0,C 180,E1 17371.345,E2 17371.345} C_VEL
LIN {X 0,Y 383.938,Z 1177.349,A -85,B 0,C 180,E1 17369.525,E2 17369.525} C_VEL
LIN {X 0,Y 382.94,Z 1177.203,A -85,B 0,C 180,E1 17368.375,E2 17368.375} C_VEL
LIN {X 0,Y 378.166,Z 1176.808,A -85,B 0,C 180,E1 17366.123,E2 17366.123} C_VEL
LIN {X 0,Y 376.134,Z 1176.19,A -85,B 0,C 180,E1 17364.712,E2 17364.712} C_VEL
LIN {X 0,Y 376.001,Z 1175.917,A -85,B 0,C 180,E1 17364.288,E2 17364.288} C_VEL
LIN {X 0,Y 376.185,Z 1172.91,A -85,B 0,C 180,E1 17360.671,E2 17360.671} C_VEL
LIN {X 0,Y 376.598,Z 1169.078,A -85,B 0,C 180,E1 17357.427,E2 17357.427} C_VEL
LIN {X 0,Y 377.335,Z 1164.36,A -85,B 0,C 180,E1 17354.321,E2 17354.321} C_VEL
LIN {X 0,Y 378.834,Z 1157.34,A -85,B 0,C 180,E1 17350.578,E2 17350.578} C_VEL
LIN {X 0,Y 381.117,Z 1148.507,A -85,B 0,C 180,E1 17346.828,E2 17346.828} C_VEL
LIN {X 0,Y 383.732,Z 1139.816,A -85,B 0,C 180,E1 17343.684,E2 17343.684} C_VEL
LIN {X 0,Y 387.798,Z 1127.956,A -85,B 0,C 180,E1 17339.989,E2 17339.989} C_VEL
LIN {X 0,Y 392.452,Z 1115.074,A -85,B 0,C 180,E1 17336.613,E2 17336.613} C_VEL
LIN {X 0,Y 397.879,Z 1101.225,A -85,B 0,C 180,E1 17333.448,E2 17333.448} C_VEL
LIN {X 0,Y 404.468,Z 1084.589,A -85,B 0,C 180,E1 17330.191,E2 17330.191} C_VEL
LIN {X 0,Y 410.998,Z 1068.446,A -85,B 0,C 180,E1 17327.446,E2 17327.446} C_VEL
LIN {X 0,Y 418.665,Z 1049.198,A -85,B 0,C 180,E1 17324.629,E2 17324.629} C_VEL
LIN {X 0,Y 425.494,Z 1031.722,A -85,B 0,C 180,E1 17322.411,E2 17322.411} C_VEL
LIN {X 0,Y 433.717,Z 1009.775,A -85,B 0,C 180,E1 17320.006,E2 17320.006} C_VEL
LIN {X 0,Y 440.013,Z 991.995,A -85,B 0,C 180,E1 17318.32,E2 17318.32} C_VEL
LIN {X 0,Y 447.299,Z 970.357,A -85,B 0,C 180,E1 17316.526,E2 17316.526} C_VEL
LIN {X 0,Y 453.962,Z 948.404,A -85,B 0,C 180,E1 17314.983,E2 17314.983} C_VEL
LIN {X 0,Y 460.645,Z 924.542,A -85,B 0,C 180,E1 17313.542,E2 17313.542} C_VEL
LIN {X 0,Y 466.36,Z 900.863,A -85,B 0,C 180,E1 17312.359,E2 17312.359} C_VEL
LIN {X 0,Y 471.713,Z 875.827,A -85,B 0,C 180,E1 17311.312,E2 17311.312} C_VEL
LIN {X 0,Y 475.977,Z 851.238,A -85,B 0,C 180,E1 17310.498,E2 17310.498} C_VEL
LIN {X 0,Y 482.168,Z 810.613,A -85,B 0,C 180,E1 17309.433,E2 17309.433} C_VEL
LIN {X 0,Y 494.273,Z 729.231,A -85,B 0,C 180,E1 17307.584,E2 17307.584} C_VEL
LIN {X 0,Y 504.447,Z 652.436,A -85,B 0,C 180,E1 17306.031,E2 17306.031} C_VEL
LIN {X 0,Y 512.472,Z 581.362,A -85,B 0,C 180,E1 17304.737,E2 17304.737} C_VEL
LIN {X 0,Y 516.817,Z 534.42,A -85,B 0,C 180,E1 17303.942,E2 17303.942} C_VEL
LIN {X 0,Y 508.321,Z 527.578,A -85,B 0,C 180,E1 17301.34,E2 17301.34} C_VEL
LIN {X 0,Y 498.862,Z 520.824,A -85,B 0,C 180,E1 17297.979,E2 17297.979} C_VEL
LIN {X 0,Y 490.29,Z 516.997,A -85,B 0,C 180,E1 17294.286,E2 17294.286} C_VEL
LIN {X 0,Y 483.909,Z 515.251,A -85,B 0,C 180,E1 17290.717,E2 17290.717} C_VEL
LIN {X 0,Y 482.068,Z 514.916,A -85,B 0,C 180,E1 17289.431,E2 17289.431} C_VEL
LIN {X 0,Y 479.566,Z 516.018,A -85,B 0,C 180,E1 17287.307,E2 17287.307} C_VEL
LIN {X 0,Y 480.652,Z 518.159,A -85,B 0,C 180,E1 17285.252,E2 17285.252} C_VEL
LIN {X 0,Y 482.25,Z 522.396,A -85,B 0,C 180,E1 17282.496,E2 17282.496} C_VEL
LIN {X 0,Y 484.007,Z 526.919,A -85,B 0,C 180,E1 17280.118,E2 17280.118} C_VEL
LIN {X 0,Y 486.495,Z 533.471,A -85,B 0,C 180,E1 17277.291,E2 17277.291} C_VEL
LIN {X 0,Y 489.756,Z 542.33,A -85,B 0,C 180,E1 17274.141,E2 17274.141} C_VEL
LIN {X 0,Y 492.108,Z 549.561,A -85,B 0,C 180,E1 17271.999,E2 17271.999} C_VEL
LIN {X 0,Y 481.801,Z 582.488,A -85,B 0,C 180,E1 17268.872,E2 17268.872} C_VEL
LIN {X 0,Y 477.434,Z 597.888,A -85,B 0,C 180,E1 17267.458,E2 17267.458} C_VEL
LIN {X 0,Y 477.956,Z 631.372,A -85,B 0,C 180,E1 17265.162,E2 17265.162} C_VEL
LIN {X 0,Y 479.229,Z 664.022,A -85,B 0,C 180,E1 17262.93,E2 17262.93} C_VEL
LIN {X 0,Y 481.388,Z 689.404,A -85,B 0,C 180,E1 17260.956,E2 17260.956} C_VEL
LIN {X 0,Y 484.202,Z 710.422,A -85,B 0,C 180,E1 17259.1,E2 17259.1} C_VEL
LIN {X 0,Y 487.346,Z 727.531,A -85,B 0,C 180,E1 17257.439,E2 17257.439} C_VEL
LIN {X 0,Y 491.298,Z 744.173,A -85,B 0,C 180,E1 17255.677,E2 17255.677} C_VEL
LIN {X 0,Y 497.484,Z 763.685,A -85,B 0,C 180,E1 17253.403,E2 17253.403} C_VEL
LIN {X 0,Y 500.062,Z 770.412,A -85,B 0,C 180,E1 17252.569,E2 17252.569} C_VEL
LIN {X 0,Y 496.869,Z 792.722,A -85,B 0,C 180,E1 17252.201,E2 17252.201} C_VEL
LIN {X 0,Y 490.416,Z 832.925,A -85,B 0,C 180,E1 17251.304,E2 17251.304} C_VEL
LIN {X 0,Y 483.559,Z 868.368,A -85,B 0,C 180,E1 17250.366,E2 17250.366} C_VEL
LIN {X 0,Y 476.586,Z 901.207,A -85,B 0,C 180,E1 17249.261,E2 17249.261} C_VEL
LIN {X 0,Y 469.429,Z 932.447,A -85,B 0,C 180,E1 17247.963,E2 17247.963} C_VEL
LIN {X 0,Y 462.276,Z 961.849,A -85,B 0,C 180,E1 17246.501,E2 17246.501} C_VEL
LIN {X 0,Y 454.706,Z 991.258,A -85,B 0,C 180,E1 17244.774,E2 17244.774} C_VEL
LIN {X 0,Y 448.262,Z 1013.742,A -85,B 0,C 180,E1 17243.201,E2 17243.201} C_VEL
LIN {X 0,Y 441.562,Z 1034.388,A -85,B 0,C 180,E1 17241.485,E2 17241.485} C_VEL
LIN {X 0,Y 434.205,Z 1055.214,A -85,B 0,C 180,E1 17239.454,E2 17239.454} C_VEL
LIN {X 0,Y 426.573,Z 1075.003,A -85,B 0,C 180,E1 17237.175,E2 17237.175} C_VEL
LIN {X 0,Y 419.119,Z 1093.074,A -85,B 0,C 180,E1 17234.728,E2 17234.728} C_VEL
LIN {X 0,Y 411.472,Z 1110.558,A -85,B 0,C 180,E1 17231.93,E2 17231.93} C_VEL
LIN {X 0,Y 404.554,Z 1125.722,A -85,B 0,C 180,E1 17229.066,E2 17229.066} C_VEL
LIN {X 0,Y 397.829,Z 1140.211,A -85,B 0,C 180,E1 17225.844,E2 17225.844} C_VEL
LIN {X 0,Y 391.646,Z 1153.737,A -85,B 0,C 180,E1 17222.245,E2 17222.245} C_VEL
LIN {X 0,Y 386.315,Z 1165.831,A -85,B 0,C 180,E1 17218.355,E2 17218.355} C_VEL
LIN {X 0,Y 382.252,Z 1175.882,A -85,B 0,C 180,E1 17214.41,E2 17214.41} C_VEL
LIN {X 0,Y 379.315,Z 1184.241,A -85,B 0,C 180,E1 17210.36,E2 17210.36} C_VEL
LIN {X 0,Y 377.392,Z 1191.085,A -85,B 0,C 180,E1 17206.15,E2 17206.15} C_VEL
LIN {X 0,Y 376.4,Z 1196.057,A -85,B 0,C 180,E1 17202.112,E2 17202.112} C_VEL
LIN {X 0,Y 376.033,Z 1199.45,A -85,B 0,C 180,E1 17198.254,E2 17198.254} C_VEL
LIN {X 0,Y 375.943,Z 1201.45,A -85,B 0,C 180,E1 17194.575,E2 17194.575} C_VEL
LIN {X 0,Y 375.947,Z 1202.276,A -85,B 0,C 180,E1 17190.912,E2 17190.912} C_VEL
LIN {X 0,Y 375.945,Z 1202.001,A -85,B 0,C 180,E1 17187.254,E2 17187.254} C_VEL
LIN {X 0,Y 375.968,Z 1200.613,A -85,B 0,C 180,E1 17183.585,E2 17183.585} C_VEL
LIN {X 0,Y 376.173,Z 1197.853,A -85,B 0,C 180,E1 17179.74,E2 17179.74} C_VEL
LIN {X 0,Y 376.851,Z 1193.571,A -85,B 0,C 180,E1 17175.713,E2 17175.713} C_VEL
LIN {X 0,Y 378.275,Z 1187.672,A -85,B 0,C 180,E1 17171.613,E2 17171.613} C_VEL
LIN {X 0,Y 380.639,Z 1180.279,A -85,B 0,C 180,E1 17167.609,E2 17167.609} C_VEL
LIN {X 0,Y 384.198,Z 1170.925,A -85,B 0,C 180,E1 17163.544,E2 17163.544} C_VEL
LIN {X 0,Y 388.981,Z 1159.69,A -85,B 0,C 180,E1 17159.574,E2 17159.574} C_VEL
LIN {X 0,Y 394.6,Z 1147.231,A -85,B 0,C 180,E1 17155.943,E2 17155.943} C_VEL
LIN {X 0,Y 401.373,Z 1132.572,A -85,B 0,C 180,E1 17152.391,E2 17152.391} C_VEL
LIN {X 0,Y 408.594,Z 1116.812,A -85,B 0,C 180,E1 17149.201,E2 17149.201} C_VEL
LIN {X 0,Y 416.105,Z 1099.966,A -85,B 0,C 180,E1 17146.328,E2 17146.328} C_VEL
LIN {X 0,Y 423.702,Z 1082.106,A -85,B 0,C 180,E1 17143.745,E2 17143.745} C_VEL
LIN {X 0,Y 431.276,Z 1063.032,A -85,B 0,C 180,E1 17141.407,E2 17141.407} C_VEL
LIN {X 0,Y 438.563,Z 1043.151,A -85,B 0,C 180,E1 17139.333,E2 17139.333} C_VEL
LIN {X 0,Y 445.765,Z 1021.679,A -85,B 0,C 180,E1 17137.433,E2 17137.433} C_VEL
LIN {X 0,Y 452.379,Z 999.581,A -85,B 0,C 180,E1 17135.788,E2 17135.788} C_VEL
LIN {X 0,Y 459.25,Z 973.737,A -85,B 0,C 180,E1 17134.172,E2 17134.172} C_VEL
LIN {X 0,Y 467.243,Z 941.527,A -85,B 0,C 180,E1 17132.465,E2 17132.465} C_VEL
LIN {X 0,Y 474.894,Z 908.442,A -85,B 0,C 180,E1 17131.024,E2 17131.024} C_VEL
LIN {X 0,Y 482.116,Z 875.031,A -85,B 0,C 180,E1 17129.843,E2 17129.843} C_VEL
LIN {X 0,Y 489.083,Z 839.909,A -85,B 0,C 180,E1 17128.869,E2 17128.869} C_VEL
LIN {X 0,Y 495.658,Z 800.523,A -85,B 0,C 180,E1 17127.968,E2 17127.968} C_VEL
LIN {X 0,Y 501.146,Z 757.999,A -85,B 0,C 180,E1 17127.153,E2 17127.153} C_VEL
LIN {X 0,Y 505.053,Z 716.614,A -85,B 0,C 180,E1 17126.521,E2 17126.521} C_VEL
LIN {X 0,Y 508.752,Z 668.434,A -85,B 0,C 180,E1 17125.882,E2 17125.882} C_VEL
LIN {X 0,Y 510.829,Z 644.126,A -85,B 0,C 180,E1 17125.522,E2 17125.522} C_VEL
LIN {X 0,Y 516.292,Z 605.804,A -85,B 0,C 180,E1 17124.942,E2 17124.942} C_VEL
LIN {X 0,Y 521.369,Z 569.428,A -85,B 0,C 180,E1 17124.368,E2 17124.368} C_VEL
LIN {X 0,Y 524.565,Z 548.233,A -85,B 0,C 180,E1 17124.087,E2 17124.087} C_VEL
LIN {X 0,Y 525.967,Z 537.284,A -85,B 0,C 180,E1 17123.886,E2 17123.886} C_VEL
LIN {X 0,Y 525.045,Z 535.682,A -85,B 0,C 180,E1 17123.603,E2 17123.603} C_VEL
LIN {X 0,Y 521.712,Z 543.711,A -85,B 0,C 180,E1 17123.224,E2 17123.224} C_VEL
LIN {X 0,Y 515.16,Z 558.927,A -85,B 0,C 180,E1 17122.42,E2 17122.42} C_VEL
LIN {X 0,Y 512.922,Z 564.19,A -85,B 0,C 180,E1 17122.138,E2 17122.138} C_VEL
LIN {X 0,Y 506.515,Z 580.083,A -85,B 0,C 180,E1 17121.344,E2 17121.344} C_VEL
LIN {X 0,Y 502.949,Z 588.422,A -85,B 0,C 180,E1 17120.854,E2 17120.854} C_VEL
LIN {X 0,Y 496.72,Z 604.612,A -85,B 0,C 180,E1 17120.05,E2 17120.05} C_VEL
LIN {X 0,Y 492.594,Z 614.568,A -85,B 0,C 180,E1 17119.445,E2 17119.445} C_VEL
LIN {X 0,Y 488.844,Z 626.706,A -85,B 0,C 180,E1 17118.878,E2 17118.878} C_VEL
LIN {X 0,Y 483.887,Z 643.481,A -85,B 0,C 180,E1 17117.901,E2 17117.901} C_VEL
LIN {X 0,Y 477.876,Z 667.781,A -85,B 0,C 180,E1 17116.799,E2 17116.799} C_VEL
LIN {X 0,Y 472.904,Z 685.629,A -85,B 0,C 180,E1 17115.765,E2 17115.765} C_VEL
LIN {X 0,Y 471.517,Z 690.625,A -85,B 0,C 180,E1 17115.497,E2 17115.497} C_VEL
LIN {X 0,Y 465.845,Z 711.368,A -85,B 0,C 180,E1 17114.502,E2 17114.502} C_VEL
LIN {X 0,Y 460.808,Z 726.925,A -85,B 0,C 180,E1 17113.512,E2 17113.512} C_VEL
LIN {X 0,Y 454.139,Z 748.456,A -85,B 0,C 180,E1 17112.396,E2 17112.396} C_VEL
LIN {X 0,Y 448.985,Z 763.014,A -85,B 0,C 180,E1 17111.405,E2 17111.405} C_VEL
LIN {X 0,Y 443.414,Z 779.547,A -85,B 0,C 180,E1 17110.487,E2 17110.487} C_VEL
LIN {X 0,Y 438.734,Z 792.087,A -85,B 0,C 180,E1 17109.569,E2 17109.569} C_VEL
LIN {X 0,Y 433.27,Z 807.451,A -85,B 0,C 180,E1 17108.652,E2 17108.652} C_VEL
LIN {X 0,Y 429.13,Z 818.179,A -85,B 0,C 180,E1 17107.806,E2 17107.806} C_VEL
LIN {X 0,Y 424.07,Z 831.964,A -85,B 0,C 180,E1 17106.944,E2 17106.944} C_VEL
LIN {X 0,Y 419.931,Z 842.468,A -85,B 0,C 180,E1 17106.07,E2 17106.07} C_VEL
LIN {X 0,Y 415.084,Z 855.507,A -85,B 0,C 180,E1 17105.209,E2 17105.209} C_VEL
LIN {X 0,Y 411.502,Z 864.695,A -85,B 0,C 180,E1 17104.39,E2 17104.39} C_VEL
LIN {X 0,Y 406.288,Z 878.849,A -85,B 0,C 180,E1 17103.527,E2 17103.527} C_VEL
LIN {X 0,Y 402.404,Z 888.955,A -85,B 0,C 180,E1 17102.689,E2 17102.689} C_VEL
LIN {X 0,Y 398.265,Z 900.442,A -85,B 0,C 180,E1 17102.235,E2 17102.235} C_VEL
LIN {X 0,Y 395.28,Z 908.467,A -85,B 0,C 180,E1 17101.667,E2 17101.667} C_VEL
LIN {X 0,Y 394.657,Z 910.161,A -85,B 0,C 180,E1 17101.55,E2 17101.55} C_VEL
LIN {X 0,Y 390.787,Z 920.349,A -85,B 0,C 180,E1 17101.136,E2 17101.136} C_VEL
LIN {X 0,Y 388.304,Z 926.652,A -85,B 0,C 180,E1 17100.664,E2 17100.664} C_VEL
LIN {X 0,Y 387.544,Z 928.905,A -85,B 0,C 180,E1 17100.43,E2 17100.43} C_VEL
LIN {X 0,Y 386.081,Z 987.644,A -85,B 0,C 180,E1 17099.022,E2 17099.022} C_VEL
LIN {X 0,Y 386.115,Z 1006.604,A -85,B 0,C 180,E1 17098.474,E2 17098.474} C_VEL
LIN {X 0,Y 385.88,Z 1021.761,A -85,B 0,C 180,E1 17097.772,E2 17097.772} C_VEL
LIN {X 0,Y 385.457,Z 1033.312,A -85,B 0,C 180,E1 17097.026,E2 17097.026} C_VEL
LIN {X 0,Y 384.914,Z 1044.226,A -85,B 0,C 180,E1 17096.127,E2 17096.127} C_VEL
LIN {X 0,Y 384.153,Z 1055.878,A -85,B 0,C 180,E1 17094.923,E2 17094.923} C_VEL
LIN {X 0,Y 383.216,Z 1066.576,A -85,B 0,C 180,E1 17093.483,E2 17093.483} C_VEL
LIN {X 0,Y 382.444,Z 1074.343,A -85,B 0,C 180,E1 17092.186,E2 17092.186} C_VEL
LIN {X 0,Y 381.694,Z 1081.056,A -85,B 0,C 180,E1 17090.805,E2 17090.805} C_VEL
LIN {X 0,Y 380.955,Z 1087.02,A -85,B 0,C 180,E1 17089.26,E2 17089.26} C_VEL
LIN {X 0,Y 380.168,Z 1092.794,A -85,B 0,C 180,E1 17087.236,E2 17087.236} C_VEL
LIN {X 0,Y 379.598,Z 1096.22,A -85,B 0,C 180,E1 17085.352,E2 17085.352} C_VEL
LIN {X 0,Y 379.239,Z 1097.986,A -85,B 0,C 180,E1 17083.684,E2 17083.684} C_VEL
LIN {X 0,Y 379.012,Z 1098.593,A -85,B 0,C 180,E1 17082.021,E2 17082.021} C_VEL
LIN {X 0,Y 378.901,Z 1098.096,A -85,B 0,C 180,E1 17080.409,E2 17080.409} C_VEL
LIN {X 0,Y 378.907,Z 1096.336,A -85,B 0,C 180,E1 17078.644,E2 17078.644} C_VEL
LIN {X 0,Y 379.102,Z 1092.563,A -85,B 0,C 180,E1 17076.53,E2 17076.53} C_VEL
LIN {X 0,Y 379.447,Z 1087.092,A -85,B 0,C 180,E1 17074.562,E2 17074.562} C_VEL
LIN {X 0,Y 379.895,Z 1081.049,A -85,B 0,C 180,E1 17072.913,E2 17072.913} C_VEL
LIN {X 0,Y 380.561,Z 1072.548,A -85,B 0,C 180,E1 17071.089,E2 17071.089} C_VEL
LIN {X 0,Y 381.293,Z 1062.391,A -85,B 0,C 180,E1 17069.42,E2 17069.42} C_VEL
LIN {X 0,Y 381.936,Z 1052.978,A -85,B 0,C 180,E1 17068.162,E2 17068.162} C_VEL
LIN {X 0,Y 382.681,Z 1040.812,A -85,B 0,C 180,E1 17066.838,E2 17066.838} C_VEL
LIN {X 0,Y 383.218,Z 1030.439,A -85,B 0,C 180,E1 17065.918,E2 17065.918} C_VEL
LIN {X 0,Y 384.618,Z 1030.87,A -85,B 0,C 180,E1 17065.477,E2 17065.477} C_VEL
LIN {X 0,Y 387.398,Z 1029.933,A -85,B 0,C 180,E1 17065.041,E2 17065.041} C_VEL
LIN {X 0,Y 391.96,Z 1028.84,A -85,B 0,C 180,E1 17064.255,E2 17064.255} C_VEL
LIN {X 0,Y 394.178,Z 1028.04,A -85,B 0,C 180,E1 17063.949,E2 17063.949} C_VEL
LIN {X 0,Y 398.465,Z 1026.679,A -85,B 0,C 180,E1 17063.328,E2 17063.328} C_VEL
LIN {X 0,Y 406.081,Z 1023.826,A -85,B 0,C 180,E1 17062.363,E2 17062.363} C_VEL
LIN {X 0,Y 415.147,Z 1019.851,A -85,B 0,C 180,E1 17061.405,E2 17061.405} C_VEL
LIN {X 0,Y 423.865,Z 1015.575,A -85,B 0,C 180,E1 17060.612,E2 17060.612} C_VEL
LIN {X 0,Y 433.509,Z 1010.214,A -85,B 0,C 180,E1 17059.859,E2 17059.859} C_VEL
LIN {X 0,Y 424.942,Z 1033.025,A -85,B 0,C 180,E1 17057.338,E2 17057.338} C_VEL
LIN {X 0,Y 417.251,Z 1052.778,A -85,B 0,C 180,E1 17054.793,E2 17054.793} C_VEL
LIN {X 0,Y 409.727,Z 1071.483,A -85,B 0,C 180,E1 17051.966,E2 17051.966} C_VEL
LIN {X 0,Y 402.757,Z 1089.001,A -85,B 0,C 180,E1 17048.912,E2 17048.912} C_VEL
LIN {X 0,Y 396.351,Z 1104.934,A -85,B 0,C 180,E1 17045.646,E2 17045.646} C_VEL
LIN {X 0,Y 391.013,Z 1119.083,A -85,B 0,C 180,E1 17042.308,E2 17042.308} C_VEL
LIN {X 0,Y 386.388,Z 1131.771,A -85,B 0,C 180,E1 17038.774,E2 17038.774} C_VEL
LIN {X 0,Y 383.072,Z 1141.906,A -85,B 0,C 180,E1 17035.512,E2 17035.512} C_VEL
LIN {X 0,Y 380.006,Z 1152.523,A -85,B 0,C 180,E1 17031.455,E2 17031.455} C_VEL
LIN {X 0,Y 378.289,Z 1159.609,A -85,B 0,C 180,E1 17028.175,E2 17028.175} C_VEL
LIN {X 0,Y 377.143,Z 1165.496,A -85,B 0,C 180,E1 17024.904,E2 17024.904} C_VEL
LIN {X 0,Y 376.379,Z 1171.013,A -85,B 0,C 180,E1 17021.029,E2 17021.029} C_VEL
LIN {X 0,Y 376.073,Z 1174.5,A -85,B 0,C 180,E1 17017.488,E2 17017.488} C_VEL
LIN {X 0,Y 375.968,Z 1176.483,A -85,B 0,C 180,E1 17014.425,E2 17014.425} C_VEL
LIN {X 0,Y 375.95,Z 1177.436,A -85,B 0,C 180,E1 17011.526,E2 17011.526} C_VEL
LIN {X 0,Y 375.949,Z 1177.498,A -85,B 0,C 180,E1 17008.783,E2 17008.783} C_VEL
LIN {X 0,Y 375.967,Z 1176.666,A -85,B 0,C 180,E1 17005.884,E2 17005.884} C_VEL
LIN {X 0,Y 376.001,Z 1175.917,A -85,B 0,C 180,E1 17004.288,E2 17004.288} C_VEL
LIN {X 0,Y 375.043,Z 1175.138,A -85,B 0,C 180,E1 17003.12,E2 17003.12} C_VEL
LIN {X 0,Y 368.812,Z 1172.477,A -85,B 0,C 180,E1 16999.826,E2 16999.826} C_VEL
LIN {X 0,Y 368.377,Z 1171.614,A -85,B 0,C 180,E1 16998.97,E2 16998.97} C_VEL
LIN {X 0,Y 369.184,Z 1166.155,A -85,B 0,C 180,E1 16994.932,E2 16994.932} C_VEL
LIN {X 0,Y 370.376,Z 1160.344,A -85,B 0,C 180,E1 16991.59,E2 16991.59} C_VEL
LIN {X 0,Y 372.063,Z 1153.692,A -85,B 0,C 180,E1 16988.399,E2 16988.399} C_VEL
LIN {X 0,Y 374.948,Z 1144.246,A -85,B 0,C 180,E1 16984.576,E2 16984.576} C_VEL
LIN {X 0,Y 378.632,Z 1133.341,A -85,B 0,C 180,E1 16980.931,E2 16980.931} C_VEL
LIN {X 0,Y 382.936,Z 1121.961,A -85,B 0,C 180,E1 16977.64,E2 16977.64} C_VEL
LIN {X 0,Y 388.897,Z 1106.933,A -85,B 0,C 180,E1 16973.932,E2 16973.932} C_VEL
LIN {X 0,Y 394.835,Z 1092.671,A -85,B 0,C 180,E1 16970.911,E2 16970.911} C_VEL
LIN {X 0,Y 402.303,Z 1074.861,A -85,B 0,C 180,E1 16967.662,E2 16967.662} C_VEL
LIN {X 0,Y 409.177,Z 1058.423,A -85,B 0,C 180,E1 16965.075,E2 16965.075} C_VEL
LIN {X 0,Y 417.6,Z 1037.824,A -85,B 0,C 180,E1 16962.284,E2 16962.284} C_VEL
LIN {X 0,Y 424.941,Z 1019.235,A -85,B 0,C 180,E1 16960.121,E2 16960.121} C_VEL
LIN {X 0,Y 433.299,Z 996.935,A -85,B 0,C 180,E1 16957.892,E2 16957.892} C_VEL
LIN {X 0,Y 440.185,Z 977.241,A -85,B 0,C 180,E1 16956.199,E2 16956.199} C_VEL
LIN {X 0,Y 447.929,Z 953.247,A -85,B 0,C 180,E1 16954.434,E2 16954.434} C_VEL
LIN {X 0,Y 454.243,Z 931.647,A -85,B 0,C 180,E1 16953.087,E2 16953.087} C_VEL
LIN {X 0,Y 460.882,Z 906.012,A -85,B 0,C 180,E1 16951.744,E2 16951.744} C_VEL
LIN {X 0,Y 465.67,Z 884.631,A -85,B 0,C 180,E1 16950.813,E2 16950.813} C_VEL
LIN {X 0,Y 470.505,Z 859.636,A -85,B 0,C 180,E1 16949.911,E2 16949.911} C_VEL
LIN {X 0,Y 476.126,Z 824.307,A -85,B 0,C 180,E1 16948.929,E2 16948.929} C_VEL
LIN {X 0,Y 488.907,Z 741.46,A -85,B 0,C 180,E1 16947.011,E2 16947.011} C_VEL
LIN {X 0,Y 499.287,Z 666.719,A -85,B 0,C 180,E1 16945.473,E2 16945.473} C_VEL
LIN {X 0,Y 507.732,Z 595.972,A -85,B 0,C 180,E1 16944.165,E2 16944.165} C_VEL
LIN {X 0,Y 513.114,Z 540.591,A -85,B 0,C 180,E1 16943.211,E2 16943.211} C_VEL
LIN {X 0,Y 506.681,Z 535.266,A -85,B 0,C 180,E1 16941.17,E2 16941.17} C_VEL
LIN {X 0,Y 497.334,Z 528.592,A -85,B 0,C 180,E1 16937.794,E2 16937.794} C_VEL
LIN {X 0,Y 489.102,Z 524.901,A -85,B 0,C 180,E1 16934.201,E2 16934.201} C_VEL
LIN {X 0,Y 482.768,Z 523.171,A -85,B 0,C 180,E1 16930.622,E2 16930.622} C_VEL
LIN {X 0,Y 481.098,Z 522.894,A -85,B 0,C 180,E1 16929.45,E2 16929.45} C_VEL
LIN {X 0,Y 476.421,Z 525.136,A -85,B 0,C 180,E1 16925.178,E2 16925.178} C_VEL
LIN {X 0,Y 477.879,Z 528.989,A -85,B 0,C 180,E1 16922.638,E2 16922.638} C_VEL
LIN {X 0,Y 479.59,Z 533.514,A -85,B 0,C 180,E1 16920.239,E2 16920.239} C_VEL
LIN {X 0,Y 482.018,Z 540.093,A -85,B 0,C 180,E1 16917.384,E2 16917.384} C_VEL
LIN {X 0,Y 485.084,Z 548.646,A -85,B 0,C 180,E1 16914.322,E2 16914.322} C_VEL
LIN {X 0,Y 487.046,Z 554.571,A -85,B 0,C 180,E1 16912.509,E2 16912.509} C_VEL
LIN {X 0,Y 476.453,Z 587.588,A -85,B 0,C 180,E1 16909.358,E2 16909.358} C_VEL
LIN {X 0,Y 475.491,Z 591.561,A -85,B 0,C 180,E1 16909.01,E2 16909.01} C_VEL
LIN {X 0,Y 475.608,Z 625.432,A -85,B 0,C 180,E1 16906.621,E2 16906.621} C_VEL
LIN {X 0,Y 476.694,Z 666.717,A -85,B 0,C 180,E1 16903.801,E2 16903.801} C_VEL
LIN {X 0,Y 478.532,Z 692.257,A -85,B 0,C 180,E1 16901.813,E2 16901.813} C_VEL
LIN {X 0,Y 481.143,Z 714.596,A -85,B 0,C 180,E1 16899.836,E2 16899.836} C_VEL
LIN {X 0,Y 484.155,Z 732.6,A -85,B 0,C 180,E1 16898.065,E2 16898.065} C_VEL
LIN {X 0,Y 487.951,Z 749.511,A -85,B 0,C 180,E1 16896.255,E2 16896.255} C_VEL
LIN {X 0,Y 493.984,Z 769.38,A -85,B 0,C 180,E1 16893.912,E2 16893.912} C_VEL
LIN {X 0,Y 495.654,Z 774.091,A -85,B 0,C 180,E1 16893.333,E2 16893.333} C_VEL
LIN {X 0,Y 491.792,Z 800.049,A -85,B 0,C 180,E1 16892.854,E2 16892.854} C_VEL
LIN {X 0,Y 485.227,Z 838.472,A -85,B 0,C 180,E1 16891.976,E2 16891.976} C_VEL
LIN {X 0,Y 478.223,Z 872.912,A -85,B 0,C 180,E1 16891.03,E2 16891.03} C_VEL
LIN {X 0,Y 470.824,Z 906.446,A -85,B 0,C 180,E1 16889.864,E2 16889.864} C_VEL
LIN {X 0,Y 463.252,Z 938.549,A -85,B 0,C 180,E1 16888.488,E2 16888.488} C_VEL
LIN {X 0,Y 455.703,Z 968.476,A -85,B 0,C 180,E1 16886.944,E2 16886.944} C_VEL
LIN {X 0,Y 448.699,Z 994.371,A -85,B 0,C 180,E1 16885.372,E2 16885.372} C_VEL
LIN {X 0,Y 442.211,Z 1016.037,A -85,B 0,C 180,E1 16883.821,E2 16883.821} C_VEL
LIN {X 0,Y 435.077,Z 1037.267,A -85,B 0,C 180,E1 16882.021,E2 16882.021} C_VEL
LIN {X 0,Y 427.494,Z 1057.636,A -85,B 0,C 180,E1 16879.968,E2 16879.968} C_VEL
LIN {X 0,Y 419.804,Z 1076.7,A -85,B 0,C 180,E1 16877.709,E2 16877.709} C_VEL
LIN {X 0,Y 411.674,Z 1095.563,A -85,B 0,C 180,E1 16875.07,E2 16875.07} C_VEL
LIN {X 0,Y 403.937,Z 1112.566,A -85,B 0,C 180,E1 16872.257,E2 16872.257} C_VEL
LIN {X 0,Y 396.654,Z 1127.99,A -85,B 0,C 180,E1 16869.248,E2 16869.248} C_VEL
LIN {X 0,Y 389.555,Z 1142.763,A -85,B 0,C 180,E1 16865.816,E2 16865.816} C_VEL
LIN {X 0,Y 383.323,Z 1155.888,A -85,B 0,C 180,E1 16862.147,E2 16862.147} C_VEL
LIN {X 0,Y 378.093,Z 1167.396,A -85,B 0,C 180,E1 16858.251,E2 16858.251} C_VEL
LIN {X 0,Y 374.089,Z 1176.978,A -85,B 0,C 180,E1 16854.293,E2 16854.293} C_VEL
LIN {X 0,Y 371.177,Z 1185.056,A -85,B 0,C 180,E1 16850.168,E2 16850.168} C_VEL
LIN {X 0,Y 369.34,Z 1191.44,A -85,B 0,C 180,E1 16846.028,E2 16846.028} C_VEL
LIN {X 0,Y 368.364,Z 1196.244,A -85,B 0,C 180,E1 16841.903,E2 16841.903} C_VEL
LIN {X 0,Y 368.021,Z 1199.472,A -85,B 0,C 180,E1 16837.963,E2 16837.963} C_VEL
LIN {X 0,Y 367.946,Z 1201.369,A -85,B 0,C 180,E1 16834.192,E2 16834.192} C_VEL
LIN {X 0,Y 367.944,Z 1202.04,A -85,B 0,C 180,E1 16830.621,E2 16830.621} C_VEL
LIN {X 0,Y 367.95,Z 1201.656,A -85,B 0,C 180,E1 16826.883,E2 16826.883} C_VEL
LIN {X 0,Y 367.978,Z 1200.155,A -85,B 0,C 180,E1 16823.132,E2 16823.132} C_VEL
LIN {X 0,Y 368.225,Z 1197.318,A -85,B 0,C 180,E1 16819.199,E2 16819.199} C_VEL
LIN {X 0,Y 369.008,Z 1192.901,A -85,B 0,C 180,E1 16815.081,E2 16815.081} C_VEL
LIN {X 0,Y 370.572,Z 1186.932,A -85,B 0,C 180,E1 16810.943,E2 16810.943} C_VEL
LIN {X 0,Y 373.225,Z 1179.218,A -85,B 0,C 180,E1 16806.769,E2 16806.769} C_VEL
LIN {X 0,Y 377.038,Z 1169.779,A -85,B 0,C 180,E1 16802.674,E2 16802.674} C_VEL
LIN {X 0,Y 381.948,Z 1158.772,A -85,B 0,C 180,E1 16798.778,E2 16798.778} C_VEL
LIN {X 0,Y 388.015,Z 1145.944,A -85,B 0,C 180,E1 16795.032,E2 16795.032} C_VEL
LIN {X 0,Y 395.01,Z 1131.319,A -85,B 0,C 180,E1 16791.485,E2 16791.485} C_VEL
LIN {X 0,Y 402.575,Z 1115.415,A -85,B 0,C 180,E1 16788.267,E2 16788.267} C_VEL
LIN {X 0,Y 410.264,Z 1098.716,A -85,B 0,C 180,E1 16785.418,E2 16785.418} C_VEL
LIN {X 0,Y 418.031,Z 1080.976,A -85,B 0,C 180,E1 16782.85,E2 16782.85} C_VEL
LIN {X 0,Y 425.928,Z 1061.634,A -85,B 0,C 180,E1 16780.481,E2 16780.481} C_VEL
LIN {X 0,Y 433.759,Z 1040.805,A -85,B 0,C 180,E1 16778.323,E2 16778.323} C_VEL
LIN {X 0,Y 441.196,Z 1019.05,A -85,B 0,C 180,E1 16776.426,E2 16776.426} C_VEL
LIN {X 0,Y 448.035,Z 996.723,A -85,B 0,C 180,E1 16774.786,E2 16774.786} C_VEL
LIN {X 0,Y 455.207,Z 970.134,A -85,B 0,C 180,E1 16773.158,E2 16773.158} C_VEL
LIN {X 0,Y 463.85,Z 935.838,A -85,B 0,C 180,E1 16771.39,E2 16771.39} C_VEL
LIN {X 0,Y 471.387,Z 903.865,A -85,B 0,C 180,E1 16770.04,E2 16770.04} C_VEL
LIN {X 0,Y 478.889,Z 869.578,A -85,B 0,C 180,E1 16768.871,E2 16768.871} C_VEL
LIN {X 0,Y 486.294,Z 832.381,A -85,B 0,C 180,E1 16767.882,E2 16767.882} C_VEL
LIN {X 0,Y 492.7,Z 793.329,A -85,B 0,C 180,E1 16767.011,E2 16767.011} C_VEL
LIN {X 0,Y 497.938,Z 752.986,A -85,B 0,C 180,E1 16766.26,E2 16766.26} C_VEL
LIN {X 0,Y 501.689,Z 714.198,A -85,B 0,C 180,E1 16765.674,E2 16765.674} C_VEL
LIN {X 0,Y 505.125,Z 670.148,A -85,B 0,C 180,E1 16765.086,E2 16765.086} C_VEL
LIN {X 0,Y 507.677,Z 640.428,A -85,B 0,C 180,E1 16764.66,E2 16764.66} C_VEL
LIN {X 0,Y 512.627,Z 606.274,A -85,B 0,C 180,E1 16764.151,E2 16764.151} C_VEL
LIN {X 0,Y 517.826,Z 569.581,A -85,B 0,C 180,E1 16763.577,E2 16763.577} C_VEL
LIN {X 0,Y 519.555,Z 558.161,A -85,B 0,C 180,E1 16763.425,E2 16763.425} C_VEL
LIN {X 0,Y 515.261,Z 567.807,A -85,B 0,C 180,E1 16762.89,E2 16762.89} C_VEL
LIN {X 0,Y 508.666,Z 583.951,A -85,B 0,C 180,E1 16762.098,E2 16762.098} C_VEL
LIN {X 0,Y 504.944,Z 592.566,A -85,B 0,C 180,E1 16761.604,E2 16761.604} C_VEL
LIN {X 0,Y 498.511,Z 608.976,A -85,B 0,C 180,E1 16760.795,E2 16760.795} C_VEL
LIN {X 0,Y 494.462,Z 618.629,A -85,B 0,C 180,E1 16760.221,E2 16760.221} C_VEL
LIN {X 0,Y 490.534,Z 631.276,A -85,B 0,C 180,E1 16759.633,E2 16759.633} C_VEL
LIN {X 0,Y 485.21,Z 649.201,A -85,B 0,C 180,E1 16758.628,E2 16758.628} C_VEL
LIN {X 0,Y 479.491,Z 671.791,A -85,B 0,C 180,E1 16757.608,E2 16757.608} C_VEL
LIN {X 0,Y 474.291,Z 689.898,A -85,B 0,C 180,E1 16756.567,E2 16756.567} C_VEL
LIN {X 0,Y 472.161,Z 697.83,A -85,B 0,C 180,E1 16756.193,E2 16756.193} C_VEL
LIN {X 0,Y 466.42,Z 717.668,A -85,B 0,C 180,E1 16755.212,E2 16755.212} C_VEL
LIN {X 0,Y 461.268,Z 733.161,A -85,B 0,C 180,E1 16754.249,E2 16754.249} C_VEL
LIN {X 0,Y 455.391,Z 751.661,A -85,B 0,C 180,E1 16753.309,E2 16753.309} C_VEL
LIN {X 0,Y 449.85,Z 766.916,A -85,B 0,C 180,E1 16752.296,E2 16752.296} C_VEL
LIN {X 0,Y 444.042,Z 783.637,A -85,B 0,C 180,E1 16751.372,E2 16751.372} C_VEL
LIN {X 0,Y 439.292,Z 795.986,A -85,B 0,C 180,E1 16750.485,E2 16750.485} C_VEL
LIN {X 0,Y 433.616,Z 811.466,A -85,B 0,C 180,E1 16749.566,E2 16749.566} C_VEL
LIN {X 0,Y 429.346,Z 822.186,A -85,B 0,C 180,E1 16748.741,E2 16748.741} C_VEL
LIN {X 0,Y 424.027,Z 836.221,A -85,B 0,C 180,E1 16747.861,E2 16747.861} C_VEL
LIN {X 0,Y 419.877,Z 846.449,A -85,B 0,C 180,E1 16747.027,E2 16747.027} C_VEL
LIN {X 0,Y 414.709,Z 859.794,A -85,B 0,C 180,E1 16746.142,E2 16746.142} C_VEL
LIN {X 0,Y 411.568,Z 867.429,A -85,B 0,C 180,E1 16745.437,E2 16745.437} C_VEL
LIN {X 0,Y 405.827,Z 882.612,A -85,B 0,C 180,E1 16744.522,E2 16744.522} C_VEL
LIN {X 0,Y 402.148,Z 891.747,A -85,B 0,C 180,E1 16743.771,E2 16743.771} C_VEL
LIN {X 0,Y 397.941,Z 903.231,A -85,B 0,C 180,E1 16743.313,E2 16743.313} C_VEL
LIN {X 0,Y 394.763,Z 911.417,A -85,B 0,C 180,E1 16742.758,E2 16742.758} C_VEL
LIN {X 0,Y 393.719,Z 914.099,A -85,B 0,C 180,E1 16742.62,E2 16742.62} C_VEL
LIN {X 0,Y 389.748,Z 924.298,A -85,B 0,C 180,E1 16742.165,E2 16742.165} C_VEL
LIN {X 0,Y 386.909,Z 931.061,A -85,B 0,C 180,E1 16741.629,E2 16741.629} C_VEL
LIN {X 0,Y 385.709,Z 933.805,A -85,B 0,C 180,E1 16741.485,E2 16741.485} C_VEL
LIN {X 0,Y 382.027,Z 942.226,A -85,B 0,C 180,E1 16741.043,E2 16741.043} C_VEL
LIN {X 0,Y 379.97,Z 946.431,A -85,B 0,C 180,E1 16740.603,E2 16740.603} C_VEL
LIN {X 0,Y 379.634,Z 947.534,A -85,B 0,C 180,E1 16740.49,E2 16740.49} C_VEL
LIN {X 0,Y 378.69,Z 995.93,A -85,B 0,C 180,E1 16739.267,E2 16739.267} C_VEL
LIN {X 0,Y 378.619,Z 1013.775,A -85,B 0,C 180,E1 16738.638,E2 16738.638} C_VEL
LIN {X 0,Y 378.305,Z 1026.537,A -85,B 0,C 180,E1 16737.955,E2 16737.955} C_VEL
LIN {X 0,Y 377.717,Z 1040.346,A -85,B 0,C 180,E1 16736.965,E2 16736.965} C_VEL
LIN {X 0,Y 376.96,Z 1052.016,A -85,B 0,C 180,E1 16735.836,E2 16735.836} C_VEL
LIN {X 0,Y 376.159,Z 1061.783,A -85,B 0,C 180,E1 16734.662,E2 16734.662} C_VEL
LIN {X 0,Y 375.35,Z 1070.18,A -85,B 0,C 180,E1 16733.422,E2 16733.422} C_VEL
LIN {X 0,Y 374.333,Z 1079.473,A -85,B 0,C 180,E1 16731.707,E2 16731.707} C_VEL
LIN {X 0,Y 373.41,Z 1086.521,A -85,B 0,C 180,E1 16729.976,E2 16729.976} C_VEL
LIN {X 0,Y 372.704,Z 1091.496,A -85,B 0,C 180,E1 16728.392,E2 16728.392} C_VEL
LIN {X 0,Y 372.119,Z 1095.224,A -85,B 0,C 180,E1 16726.797,E2 16726.797} C_VEL
LIN {X 0,Y 371.656,Z 1097.805,A -85,B 0,C 180,E1 16725.192,E2 16725.192} C_VEL
LIN {X 0,Y 371.288,Z 1099.406,A -85,B 0,C 180,E1 16723.413,E2 16723.413} C_VEL
LIN {X 0,Y 371.04,Z 1099.713,A -85,B 0,C 180,E1 16721.296,E2 16721.296} C_VEL
LIN {X 0,Y 370.966,Z 1098.067,A -85,B 0,C 180,E1 16719.158,E2 16719.158} C_VEL
LIN {X 0,Y 371.045,Z 1095.602,A -85,B 0,C 180,E1 16717.501,E2 16717.501} C_VEL
LIN {X 0,Y 371.263,Z 1091.967,A -85,B 0,C 180,E1 16715.835,E2 16715.835} C_VEL
LIN {X 0,Y 371.605,Z 1087.052,A -85,B 0,C 180,E1 16714.157,E2 16714.157} C_VEL
LIN {X 0,Y 372.161,Z 1080.017,A -85,B 0,C 180,E1 16712.302,E2 16712.302} C_VEL
LIN {X 0,Y 372.876,Z 1070.638,A -85,B 0,C 180,E1 16710.435,E2 16710.435} C_VEL
LIN {X 0,Y 373.601,Z 1060.965,A -85,B 0,C 180,E1 16708.9,E2 16708.9} C_VEL
LIN {X 0,Y 374.44,Z 1048.737,A -85,B 0,C 180,E1 16707.356,E2 16707.356} C_VEL
LIN {X 0,Y 375.094,Z 1037.358,A -85,B 0,C 180,E1 16706.211,E2 16706.211} C_VEL
LIN {X 0,Y 376.527,Z 1037.845,A -85,B 0,C 180,E1 16705.738,E2 16705.738} C_VEL
LIN {X 0,Y 379.82,Z 1036.962,A -85,B 0,C 180,E1 16705.162,E2 16705.162} C_VEL
LIN {X 0,Y 382.893,Z 1036.449,A -85,B 0,C 180,E1 16704.568,E2 16704.568} C_VEL
LIN {X 0,Y 385.631,Z 1035.669,A -85,B 0,C 180,E1 16704.127,E2 16704.127} C_VEL
LIN {X 0,Y 390.595,Z 1034.149,A -85,B 0,C 180,E1 16703.383,E2 16703.383} C_VEL
LIN {X 0,Y 396.42,Z 1032.31,A -85,B 0,C 180,E1 16702.564,E2 16702.564} C_VEL
LIN {X 0,Y 404.138,Z 1029.493,A -85,B 0,C 180,E1 16701.61,E2 16701.61} C_VEL
LIN {X 0,Y 413.287,Z 1025.571,A -85,B 0,C 180,E1 16700.663,E2 16700.663} C_VEL
LIN {X 0,Y 423.015,Z 1020.906,A -85,B 0,C 180,E1 16699.812,E2 16699.812} C_VEL
LIN {X 0,Y 424.538,Z 1020.172,A -85,B 0,C 180,E1 16699.682,E2 16699.682} C_VEL
LIN {X 0,Y 416.486,Z 1040.577,A -85,B 0,C 180,E1 16697.278,E2 16697.278} C_VEL
LIN {X 0,Y 408.564,Z 1059.809,A -85,B 0,C 180,E1 16694.62,E2 16694.62} C_VEL
LIN {X 0,Y 401.312,Z 1077.247,A -85,B 0,C 180,E1 16691.843,E2 16691.843} C_VEL
LIN {X 0,Y 394.03,Z 1094.486,A -85,B 0,C 180,E1 16688.629,E2 16688.629} C_VEL
LIN {X 0,Y 387.965,Z 1109.271,A -85,B 0,C 180,E1 16685.444,E2 16685.444} C_VEL
LIN {X 0,Y 382.371,Z 1123.323,A -85,B 0,C 180,E1 16681.887,E2 16681.887} C_VEL
LIN {X 0,Y 378.259,Z 1134.397,A -85,B 0,C 180,E1 16678.644,E2 16678.644} C_VEL
LIN {X 0,Y 374.339,Z 1146.067,A -85,B 0,C 180,E1 16674.627,E2 16674.627} C_VEL
LIN {X 0,Y 371.925,Z 1154.19,A -85,B 0,C 180,E1 16671.282,E2 16671.282} C_VEL
LIN {X 0,Y 370.21,Z 1161.08,A -85,B 0,C 180,E1 16667.934,E2 16667.934} C_VEL
LIN {X 0,Y 368.929,Z 1167.728,A -85,B 0,C 180,E1 16663.96,E2 16663.96} C_VEL
LIN {X 0,Y 368.302,Z 1172.248,A -85,B 0,C 180,E1 16660.324,E2 16660.324} C_VEL
LIN {X 0,Y 368.06,Z 1175.107,A -85,B 0,C 180,E1 16657.181,E2 16657.181} C_VEL
LIN {X 0,Y 367.972,Z 1176.884,A -85,B 0,C 180,E1 16654.209,E2 16654.209} C_VEL
LIN {X 0,Y 367.954,Z 1177.746,A -85,B 0,C 180,E1 16651.248,E2 16651.248} C_VEL
LIN {X 0,Y 367.954,Z 1177.69,A -85,B 0,C 180,E1 16648.289,E2 16648.289} C_VEL
LIN {X 0,Y 367.979,Z 1176.717,A -85,B 0,C 180,E1 16645.326,E2 16645.326} C_VEL
LIN {X 0,Y 368.098,Z 1174.597,A -85,B 0,C 180,E1 16642.039,E2 16642.039} C_VEL
LIN {X 0,Y 368.377,Z 1171.614,A -85,B 0,C 180,E1 16638.97,E2 16638.97} C_VEL
LIN {X 0,Y 367.558,Z 1170.343,A -85,B 0,C 180,E1 16637.785,E2 16637.785} C_VEL
LIN {X 0,Y 361.953,Z 1166.244,A -85,B 0,C 180,E1 16634.53,E2 16634.53} C_VEL
LIN {X 0,Y 361.623,Z 1164.805,A -85,B 0,C 180,E1 16633.586,E2 16633.586} C_VEL
LIN {X 0,Y 363.426,Z 1157.489,A -85,B 0,C 180,E1 16629.551,E2 16629.551} C_VEL
LIN {X 0,Y 365.923,Z 1148.987,A -85,B 0,C 180,E1 16625.805,E2 16625.805} C_VEL
LIN {X 0,Y 369.037,Z 1139.925,A -85,B 0,C 180,E1 16622.401,E2 16622.401} C_VEL
LIN {X 0,Y 374.078,Z 1126.676,A -85,B 0,C 180,E1 16618.212,E2 16618.212} C_VEL
LIN {X 0,Y 378.899,Z 1114.966,A -85,B 0,C 180,E1 16615.068,E2 16615.068} C_VEL
LIN {X 0,Y 385.481,Z 1099.612,A -85,B 0,C 180,E1 16611.502,E2 16611.502} C_VEL
LIN {X 0,Y 392.151,Z 1084.323,A -85,B 0,C 180,E1 16608.479,E2 16608.479} C_VEL
LIN {X 0,Y 399.992,Z 1066.546,A -85,B 0,C 180,E1 16605.434,E2 16605.434} C_VEL
LIN {X 0,Y 407.404,Z 1049.237,A -85,B 0,C 180,E1 16602.898,E2 16602.898} C_VEL
LIN {X 0,Y 415.384,Z 1030.363,A -85,B 0,C 180,E1 16600.482,E2 16600.482} C_VEL
LIN {X 0,Y 423.683,Z 1009.324,A -85,B 0,C 180,E1 16598.194,E2 16598.194} C_VEL
LIN {X 0,Y 431.75,Z 988.027,A -85,B 0,C 180,E1 16596.197,E2 16596.197} C_VEL
LIN {X 0,Y 439.14,Z 966.574,A -85,B 0,C 180,E1 16594.492,E2 16594.492} C_VEL
LIN {X 0,Y 446.295,Z 944.315,A -85,B 0,C 180,E1 16592.966,E2 16592.966} C_VEL
LIN {X 0,Y 452.736,Z 921.326,A -85,B 0,C 180,E1 16591.641,E2 16591.641} C_VEL
LIN {X 0,Y 458.516,Z 898.611,A -85,B 0,C 180,E1 16590.533,E2 16590.533} C_VEL
LIN {X 0,Y 463.8,Z 873.872,A -85,B 0,C 180,E1 16589.543,E2 16589.543} C_VEL
LIN {X 0,Y 467.894,Z 851.284,A -85,B 0,C 180,E1 16588.805,E2 16588.805} C_VEL
LIN {X 0,Y 475.205,Z 806.439,A -85,B 0,C 180,E1 16587.642,E2 16587.642} C_VEL
LIN {X 0,Y 487.431,Z 727.925,A -85,B 0,C 180,E1 16585.869,E2 16585.869} C_VEL
LIN {X 0,Y 497.457,Z 655.918,A -85,B 0,C 180,E1 16584.418,E2 16584.418} C_VEL
LIN {X 0,Y 505.613,Z 586.943,A -85,B 0,C 180,E1 16583.168,E2 16583.168} C_VEL
LIN {X 0,Y 509.5,Z 546.723,A -85,B 0,C 180,E1 16582.47,E2 16582.47} C_VEL
LIN {X 0,Y 505.034,Z 542.953,A -85,B 0,C 180,E1 16580.999,E2 16580.999} C_VEL
LIN {X 0,Y 496.099,Z 536.469,A -85,B 0,C 180,E1 16577.719,E2 16577.719} C_VEL
LIN {X 0,Y 487.911,Z 532.802,A -85,B 0,C 180,E1 16574.115,E2 16574.115} C_VEL
LIN {X 0,Y 481.806,Z 531.112,A -85,B 0,C 180,E1 16570.644,E2 16570.644} C_VEL
LIN {X 0,Y 480.129,Z 530.869,A -85,B 0,C 180,E1 16569.469,E2 16569.469} C_VEL
LIN {X 0,Y 475.5,Z 533.015,A -85,B 0,C 180,E1 16565.309,E2 16565.309} C_VEL
LIN {X 0,Y 473.712,Z 536.251,A -85,B 0,C 180,E1 16562.419,E2 16562.419} C_VEL
LIN {X 0,Y 475.175,Z 540.11,A -85,B 0,C 180,E1 16560.362,E2 16560.362} C_VEL
LIN {X 0,Y 477.651,Z 547.014,A -85,B 0,C 180,E1 16557.36,E2 16557.36} C_VEL
LIN {X 0,Y 480.529,Z 555.337,A -85,B 0,C 180,E1 16554.388,E2 16554.388} C_VEL
LIN {X 0,Y 481.958,Z 559.833,A -85,B 0,C 180,E1 16552.999,E2 16552.999} C_VEL
LIN {X 0,Y 473.874,Z 584.84,A -85,B 0,C 180,E1 16550.627,E2 16550.627} C_VEL
LIN {X 0,Y 473.549,Z 617.767,A -85,B 0,C 180,E1 16548.228,E2 16548.228} C_VEL
LIN {X 0,Y 474.296,Z 670.879,A -85,B 0,C 180,E1 16544.572,E2 16544.572} C_VEL
LIN {X 0,Y 475.78,Z 696.154,A -85,B 0,C 180,E1 16542.587,E2 16542.587} C_VEL
LIN {X 0,Y 478.126,Z 719.055,A -85,B 0,C 180,E1 16540.547,E2 16540.547} C_VEL
LIN {X 0,Y 481.008,Z 737.664,A -85,B 0,C 180,E1 16538.699,E2 16538.699} C_VEL
LIN {X 0,Y 484.625,Z 754.959,A -85,B 0,C 180,E1 16536.824,E2 16536.824} C_VEL
LIN {X 0,Y 490.38,Z 774.939,A -85,B 0,C 180,E1 16534.437,E2 16534.437} C_VEL
LIN {X 0,Y 491.259,Z 777.798,A -85,B 0,C 180,E1 16534.099,E2 16534.099} C_VEL
LIN {X 0,Y 485.941,Z 811.933,A -85,B 0,C 180,E1 16533.414,E2 16533.414} C_VEL
LIN {X 0,Y 478.785,Z 850.196,A -85,B 0,C 180,E1 16532.499,E2 16532.499} C_VEL
LIN {X 0,Y 471.635,Z 883.561,A -85,B 0,C 180,E1 16531.509,E2 16531.509} C_VEL
LIN {X 0,Y 463.812,Z 917.299,A -85,B 0,C 180,E1 16530.251,E2 16530.251} C_VEL
LIN {X 0,Y 456.168,Z 948.101,A -85,B 0,C 180,E1 16528.849,E2 16528.849} C_VEL
LIN {X 0,Y 448.324,Z 977.979,A -85,B 0,C 180,E1 16527.222,E2 16527.222} C_VEL
LIN {X 0,Y 441.64,Z 1001.343,A -85,B 0,C 180,E1 16525.724,E2 16525.724} C_VEL
LIN {X 0,Y 434.906,Z 1022.357,A -85,B 0,C 180,E1 16524.134,E2 16524.134} C_VEL
LIN {X 0,Y 427.623,Z 1042.515,A -85,B 0,C 180,E1 16522.322,E2 16522.322} C_VEL
LIN {X 0,Y 419.965,Z 1062.01,A -85,B 0,C 180,E1 16520.263,E2 16520.263} C_VEL
LIN {X 0,Y 412.506,Z 1079.772,A -85,B 0,C 180,E1 16518.083,E2 16518.083} C_VEL
LIN {X 0,Y 404.534,Z 1097.463,A -85,B 0,C 180,E1 16515.522,E2 16515.522} C_VEL
LIN {X 0,Y 396.657,Z 1114.045,A -85,B 0,C 180,E1 16512.692,E2 16512.692} C_VEL
LIN {X 0,Y 388.97,Z 1129.66,A -85,B 0,C 180,E1 16509.539,E2 16509.539} C_VEL
LIN {X 0,Y 381.836,Z 1143.957,A -85,B 0,C 180,E1 16506.097,E2 16506.097} C_VEL
LIN {X 0,Y 375.715,Z 1156.392,A -85,B 0,C 180,E1 16502.516,E2 16502.516} C_VEL
LIN {X 0,Y 370.524,Z 1167.412,A -85,B 0,C 180,E1 16498.705,E2 16498.705} C_VEL
LIN {X 0,Y 366.223,Z 1177.309,A -85,B 0,C 180,E1 16494.517,E2 16494.517} C_VEL
LIN {X 0,Y 363.119,Z 1185.609,A -85,B 0,C 180,E1 16490.118,E2 16490.118} C_VEL
LIN {X 0,Y 361.236,Z 1192.025,A -85,B 0,C 180,E1 16485.737,E2 16485.737} C_VEL
LIN {X 0,Y 360.306,Z 1196.596,A -85,B 0,C 180,E1 16481.524,E2 16481.524} C_VEL
LIN {X 0,Y 360.009,Z 1199.594,A -85,B 0,C 180,E1 16477.499,E2 16477.499} C_VEL
LIN {X 0,Y 359.952,Z 1201.267,A -85,B 0,C 180,E1 16473.661,E2 16473.661} C_VEL
LIN {X 0,Y 359.955,Z 1201.817,A -85,B 0,C 180,E1 16469.839,E2 16469.839} C_VEL
LIN {X 0,Y 359.951,Z 1201.224,A -85,B 0,C 180,E1 16466.175,E2 16466.175} C_VEL
LIN {X 0,Y 360.01,Z 1199.493,A -85,B 0,C 180,E1 16462.337,E2 16462.337} C_VEL
LIN {X 0,Y 360.328,Z 1196.433,A -85,B 0,C 180,E1 16458.311,E2 16458.311} C_VEL
LIN {X 0,Y 361.29,Z 1191.797,A -85,B 0,C 180,E1 16454.097,E2 16454.097} C_VEL
LIN {X 0,Y 363.224,Z 1185.294,A -85,B 0,C 180,E1 16449.703,E2 16449.703} C_VEL
LIN {X 0,Y 366.338,Z 1177.017,A -85,B 0,C 180,E1 16445.354,E2 16445.354} C_VEL
LIN {X 0,Y 370.719,Z 1166.972,A -85,B 0,C 180,E1 16441.13,E2 16441.13} C_VEL
LIN {X 0,Y 376.331,Z 1155.179,A -85,B 0,C 180,E1 16437.098,E2 16437.098} C_VEL
LIN {X 0,Y 382.717,Z 1142.191,A -85,B 0,C 180,E1 16433.438,E2 16433.438} C_VEL
LIN {X 0,Y 389.864,Z 1127.867,A -85,B 0,C 180,E1 16430.072,E2 16430.072} C_VEL
LIN {X 0,Y 397.426,Z 1112.405,A -85,B 0,C 180,E1 16427.013,E2 16427.013} C_VEL
LIN {X 0,Y 405.493,Z 1095.264,A -85,B 0,C 180,E1 16424.145,E2 16424.145} C_VEL
LIN {X 0,Y 413.574,Z 1077.174,A -85,B 0,C 180,E1 16421.583,E2 16421.583} C_VEL
LIN {X 0,Y 421.901,Z 1057.227,A -85,B 0,C 180,E1 16419.195,E2 16419.195} C_VEL
LIN {X 0,Y 429.913,Z 1036.244,A -85,B 0,C 180,E1 16417.083,E2 16417.083} C_VEL
LIN {X 0,Y 437.55,Z 1014.144,A -85,B 0,C 180,E1 16415.217,E2 16415.217} C_VEL
LIN {X 0,Y 444.584,Z 991.155,A -85,B 0,C 180,E1 16413.592,E2 16413.592} C_VEL
LIN {X 0,Y 453.223,Z 959.326,A -85,B 0,C 180,E1 16411.735,E2 16411.735} C_VEL
LIN {X 0,Y 461.442,Z 926.946,A -85,B 0,C 180,E1 16410.163,E2 16410.163} C_VEL
LIN {X 0,Y 469.214,Z 893.985,A -85,B 0,C 180,E1 16408.855,E2 16408.855} C_VEL
LIN {X 0,Y 476.97,Z 858.534,A -85,B 0,C 180,E1 16407.732,E2 16407.732} C_VEL
LIN {X 0,Y 484.49,Z 819.943,A -85,B 0,C 180,E1 16406.773,E2 16406.773} C_VEL
LIN {X 0,Y 490.913,Z 778.866,A -85,B 0,C 180,E1 16405.898,E2 16405.898} C_VEL
LIN {X 0,Y 496.267,Z 734.371,A -85,B 0,C 180,E1 16405.124,E2 16405.124} C_VEL
LIN {X 0,Y 500.019,Z 690.675,A -85,B 0,C 180,E1 16404.503,E2 16404.503} C_VEL
LIN {X 0,Y 502.779,Z 656.973,A -85,B 0,C 180,E1 16404.074,E2 16404.074} C_VEL
LIN {X 0,Y 504.767,Z 635.912,A -85,B 0,C 180,E1 16403.777,E2 16403.777} C_VEL
LIN {X 0,Y 509.045,Z 606.873,A -85,B 0,C 180,E1 16403.351,E2 16403.351} C_VEL
LIN {X 0,Y 511.96,Z 585.4,A -85,B 0,C 180,E1 16402.978,E2 16402.978} C_VEL
LIN {X 0,Y 507.047,Z 596.65,A -85,B 0,C 180,E1 16402.351,E2 16402.351} C_VEL
LIN {X 0,Y 500.386,Z 613.338,A -85,B 0,C 180,E1 16401.534,E2 16401.534} C_VEL
LIN {X 0,Y 496.439,Z 622.635,A -85,B 0,C 180,E1 16400.994,E2 16400.994} C_VEL
LIN {X 0,Y 492.181,Z 636.273,A -85,B 0,C 180,E1 16400.359,E2 16400.359} C_VEL
LIN {X 0,Y 487.172,Z 652.76,A -85,B 0,C 180,E1 16399.444,E2 16399.444} C_VEL
LIN {X 0,Y 481.237,Z 675.669,A -85,B 0,C 180,E1 16398.418,E2 16398.418} C_VEL
LIN {X 0,Y 475.837,Z 693.961,A -85,B 0,C 180,E1 16397.377,E2 16397.377} C_VEL
LIN {X 0,Y 468.651,Z 719.016,A -85,B 0,C 180,E1 16396.192,E2 16396.192} C_VEL
LIN {X 0,Y 462.548,Z 737.104,A -85,B 0,C 180,E1 16395.107,E2 16395.107} C_VEL
LIN {X 0,Y 456.388,Z 755.904,A -85,B 0,C 180,E1 16394.156,E2 16394.156} C_VEL
LIN {X 0,Y 450.84,Z 770.795,A -85,B 0,C 180,E1 16393.184,E2 16393.184} C_VEL
LIN {X 0,Y 444.795,Z 787.68,A -85,B 0,C 180,E1 16392.257,E2 16392.257} C_VEL
LIN {X 0,Y 439.941,Z 799.942,A -85,B 0,C 180,E1 16391.395,E2 16391.395} C_VEL
LIN {X 0,Y 433.978,Z 815.712,A -85,B 0,C 180,E1 16390.462,E2 16390.462} C_VEL
LIN {X 0,Y 429.674,Z 826.179,A -85,B 0,C 180,E1 16389.673,E2 16389.673} C_VEL
LIN {X 0,Y 424.12,Z 840.36,A -85,B 0,C 180,E1 16388.787,E2 16388.787} C_VEL
LIN {X 0,Y 419.923,Z 850.427,A -85,B 0,C 180,E1 16387.984,E2 16387.984} C_VEL
LIN {X 0,Y 414.758,Z 863.377,A -85,B 0,C 180,E1 16387.132,E2 16387.132} C_VEL
LIN {X 0,Y 411.314,Z 871.357,A -85,B 0,C 180,E1 16386.421,E2 16386.421} C_VEL
LIN {X 0,Y 405.417,Z 886.356,A -85,B 0,C 180,E1 16385.52,E2 16385.52} C_VEL
LIN {X 0,Y 401.688,Z 895.484,A -85,B 0,C 180,E1 16384.823,E2 16384.823} C_VEL
LIN {X 0,Y 397.08,Z 907.703,A -85,B 0,C 180,E1 16384.301,E2 16384.301} C_VEL
LIN {X 0,Y 393.551,Z 916.365,A -85,B 0,C 180,E1 16383.74,E2 16383.74} C_VEL
LIN {X 0,Y 389.613,Z 926.333,A -85,B 0,C 180,E1 16383.31,E2 16383.31} C_VEL
LIN {X 0,Y 386.277,Z 933.951,A -85,B 0,C 180,E1 16382.752,E2 16382.752} C_VEL
LIN {X 0,Y 384.856,Z 937.147,A -85,B 0,C 180,E1 16382.586,E2 16382.586} C_VEL
LIN {X 0,Y 380.907,Z 945.79,A -85,B 0,C 180,E1 16382.106,E2 16382.106} C_VEL
LIN {X 0,Y 378.376,Z 950.778,A -85,B 0,C 180,E1 16381.623,E2 16381.623} C_VEL
LIN {X 0,Y 374.624,Z 958.395,A -85,B 0,C 180,E1 16381.224,E2 16381.224} C_VEL
LIN {X 0,Y 372.345,Z 962.523,A -85,B 0,C 180,E1 16380.769,E2 16380.769} C_VEL
LIN {X 0,Y 371.843,Z 963.755,A -85,B 0,C 180,E1 16380.607,E2 16380.607} C_VEL
LIN {X 0,Y 371.352,Z 1004.633,A -85,B 0,C 180,E1 16379.499,E2 16379.499} C_VEL
LIN {X 0,Y 371.181,Z 1018.106,A -85,B 0,C 180,E1 16378.929,E2 16378.929} C_VEL
LIN {X 0,Y 370.711,Z 1032.527,A -85,B 0,C 180,E1 16378.068,E2 16378.068} C_VEL
LIN {X 0,Y 369.966,Z 1045.638,A -85,B 0,C 180,E1 16376.979,E2 16376.979} C_VEL
LIN {X 0,Y 369.213,Z 1056.128,A -85,B 0,C 180,E1 16375.885,E2 16375.885} C_VEL
LIN {X 0,Y 368.181,Z 1067.474,A -85,B 0,C 180,E1 16374.389,E2 16374.389} C_VEL
LIN {X 0,Y 367.233,Z 1075.88,A -85,B 0,C 180,E1 16372.962,E2 16372.962} C_VEL
LIN {X 0,Y 366.369,Z 1082.725,A -85,B 0,C 180,E1 16371.525,E2 16371.525} C_VEL
LIN {X 0,Y 365.543,Z 1088.592,A -85,B 0,C 180,E1 16369.98,E2 16369.98} C_VEL
